// TIA Portal project "Aski-Otomasyonv2.2" (V16)

(* hardware
DEVICE "S71500/ET200MP station_1"  S7-1500 station
   slot 0: "Rail_0"  Rack  6ES7 590-1***0-0AA0
   slot 1: "PLC_8"  CPU 1511-1 PN  6ES7 511-1AK02-0AB0  V2.8
      slot 3: "CPU display_1"  6ES7591-1AA00-0AA0
      slot 32768: "PROFINET interface_1"  X1
         slot 32769: "Port_1"  X1 P1
         slot 32770: "Port_2"  X1 P2
      slot 34817: "Virtual CP interface port_1"  Virtual CP interface port  Virtual CP interface port
DEVICE "HMI_3"  KTP900 Basic PN
   slot 0: "HMI_3"  KTP900 Basic PN  6AV2 123-2JB03-0AX0  16.0.0.0
   slot 1: "HMI_RT_1"  KTP900 Basic PN  6AV2 123-2JB03-0AX0  16.0.0.0
   slot 5: "HMI_3.IE_CP_1"  PROFINET Interface  16.0.0.0
      slot 1: "PROFINET Interface_1"  PROFINET Interface
         slot 1: "Port_1"  Port
*)

// ===== PLC "PLC_8"  CPU 1511-1 PN =====

VAR_GLOBAL   // PLC tag table "Default tag table"
   "Start" AT %I0.0 : Bool;
   "Stop" AT %I0.1 : Bool;
   "sensor-HamSuKazan-alt" AT %I0.2 : Bool;
   "sensor-HamSuKazan-ust" AT %I0.3 : Bool;
   "sensor-TemizSuKazan-alt" AT %I0.4 : Bool;
   "sensor-TemizSuKazan-ust" AT %I0.5 : Bool;
   "aritmaMotor0" AT %Q0.0 : Bool;
   "aritmaMotor1" AT %Q0.1 : Bool;
   "aritmaMotor2" AT %Q0.2 : Bool;
   "motor-hamsu" AT %Q0.3 : Bool;
   "vana1-aritma0" AT %Q0.4 : Bool;
   "vana2-aritma0" AT %Q0.5 : Bool;
   "vana3-aritma0" AT %Q0.6 : Bool;
   "vana4-aritma0" AT %Q0.7 : Bool;
   "vana5-aritma0" AT %Q1.0 : Bool;
   "vana1-aritma1" AT %Q1.1 : Bool;
   "vana2-aritma1" AT %Q1.2 : Bool;
   "vana3-aritma1" AT %Q1.3 : Bool;
   "vana4-aritma1" AT %Q1.4 : Bool;
   "vana5-aritma1" AT %Q1.5 : Bool;
   "TimerTersYikama-aritma0" AT %T10 : Timer;
   "TimerDurulama-aritma0" AT %T11 : Timer;
   "Sistem" AT %Q1.6 : Bool;
   "TimerAritmaVana-aritma0" AT %T14 : Timer;
   "TimerTersYikamaVana-aritma0" AT %T15 : Timer;
   "TimerDurulamaVana-aritma0" AT %T16 : Timer;
   "TimerBypassVana-aritma0" AT %T17 : Timer;
   "TimerAritma-aritma0" AT %T18 : Timer;
   "sensor-SuCikisiVar" AT %I0.6 : Bool;
   "TimerMotor0Ariza" AT %T19 : Timer;
   "TimerMotor1Ariza" AT %T20 : Timer;
   "TimerMotor2Ariza" AT %T21 : Timer;
   "TimerAritmaVana-aritma1" AT %T22 : Timer;
   "TimerTersYikamaVana-aritma1" AT %T23 : Timer;
   "TimerDurulamaVana-aritma1" AT %T24 : Timer;
   "TimerBypassVana-aritma1" AT %T25 : Timer;
   "kuyuMotor" AT %I0.7 : Bool;
END_VAR

DATA_BLOCK "DBARITMA"   // DB1
{ S7_Optimized_Access := 'FALSE' }
VERSION : 0.1
   VAR
      "sure-Aritma" : S5Time := S5T#60s;
      "sure-TersYikama" : S5Time := S5T#20s;
      "sure-Durulama" : S5Time := S5T#10s;
      "sure-VanaDurumDegistirme" : S5Time := S5T#5s;
      "sure-MotorDegis" : Time := T#80s;
      "sure-MotorArizayaGec" : S5Time := S5T#5s;
      tesisDurumu : Byte := 0;
      toplamAritmaSayisi : Byte := 2;
      aritma0VanaKontrolDurum : Byte;
      aritma1VanaKontrolDurum : Byte;
      aritma0MotorCalisiyor : Bool;
      aritma1MotorCalisiyor : Bool;
      aritmaMotorCalisiyor : Bool;
      kalanZamanAritma : S5Time;
      kalanZamanTersYikama : S5Time;
      kalanZamanDurulama : S5Time;
      aritmaYapiliyor : Bool;
      tersYikamaYapiliyor : Bool;
      durulamaYapiliyor : Bool;
      aritmaMotor0Durum : Byte;
      aritmaMotor1Durum : Byte;
      aritmaMotor2Durum : Byte;
      kuyuMotorDurum : Byte := 0;
      durumKalanSure : Word := 1;
      temizsuSeviye : Byte := 45;
      hamsuSeviye : Byte := 92;
      arizaDurumu : Byte := 0;
      Adi : String := 'Deneme Tesis';
      temizsuDepoDoldur : Bool;
      "hmi-start" : Bool;
      "hmi-stop" : Bool;
      "hmi-aritmaSure" : Byte;
      "hmi-TersYikamaSure" : Byte;
      "hmi-DurulamaSure" : Byte;
      "hmi-VanaBeklemeSure" : Byte;
      "hmi-YaslandirmaSure" : Byte := 20;
      "hmi-TersYikamaYap" : Bool;
   END_VAR
BEGIN
END_DATA_BLOCK

DATA_BLOCK "FB-aritma0VanaKontrol_DB"   // DB2
{ S7_Optimized_Access := 'TRUE' }
VERSION : 0.1
// stored: InstanceOfName FB-aritmaVanaKontrol
"FB-aritmaVanaKontrol"
BEGIN
END_DATA_BLOCK

DATA_BLOCK "sistemDurum-Zamanlayici_DB"   // DB3
{ S7_Optimized_Access := 'TRUE' }
VERSION : 0.1
// stored: InstanceOfName aritmaDurum-Zamanlayici
"aritmaDurum-Zamanlayici"
BEGIN
END_DATA_BLOCK

DATA_BLOCK "aritmaMotorKontrol-Yaslandirma-Ariza_DB"   // DB4
{ S7_Optimized_Access := 'TRUE' }
VERSION : 0.1
// stored: InstanceOfName aritmaMotorKontrol-Yaslandirma-Ariza
"aritmaMotorKontrol-Yaslandirma-Ariza"
BEGIN
END_DATA_BLOCK

DATA_BLOCK "FB-aritma1VanaKontrol_DB"   // DB6
{ S7_Optimized_Access := 'TRUE' }
VERSION : 0.1
// stored: InstanceOfName FB-aritmaVanaKontrol
"FB-aritmaVanaKontrol"
BEGIN
END_DATA_BLOCK

DATA_BLOCK "TemizSuDepoSeviyeKonrolcusu"   // DB7
{ S7_Optimized_Access := 'TRUE' }
VERSION : 0.1
// stored: InstanceOfName depoSeviyeKonrolcusu
"depoSeviyeKonrolcusu"
BEGIN
END_DATA_BLOCK

DATA_BLOCK "HamSuDepoSeviyeKonrolcusu"   // DB8
{ S7_Optimized_Access := 'TRUE' }
VERSION : 0.1
// stored: InstanceOfName depoSeviyeKonrolcusu
"depoSeviyeKonrolcusu"
BEGIN
END_DATA_BLOCK

// folder: System blocks/Program resources

DATA_BLOCK "timerMotorDegistirme"   // DB5
{ S7_Optimized_Access := 'TRUE' }
AUTHOR : Simatic
FAMILY : IEC
NAME : IEC_TMR
VERSION : 1.0
// stored: InstanceOfName IEC_TIMER
"IEC_TIMER"
BEGIN
END_DATA_BLOCK

// folder: (top level)

FUNCTION_BLOCK "FB-aritmaVanaKontrol"   // FB1, LAD
{ S7_Optimized_Access := 'TRUE' }
VERSION : 0.1
   VAR_INPUT
      Sistem : Bool;
      timerAritmaVana : Timer;
      timerTersYikamaVana : Timer;
      timerDurulamaVana : Timer;
      timerBypassVana : Timer;
      "sure-VanaDurumDegisim" : S5Time;
      aritmaDurumu : Byte;
   END_VAR
   VAR_OUTPUT
      V1 : Bool;
      V2 : Bool;
      V3 : Bool;
      V4 : Bool;
      V5 : Bool;
      "aritma-motoru-Calistir" : Bool;
   END_VAR
   VAR
      aritmaDurumunaGec : Bool;
      tersYikamaDurumunaGec : Bool;
      durulamaDurumunaGec : Bool;
      bypassDurumunaGec : Bool;
      "motoruAktifEt-Aritma" : Bool;
      "motoruAktifEt-TersYikama" : Bool;
      "motoruAktifEt-Durulama" : Bool;
      "motoruAktifEt-Bypass" : Bool;
   END_VAR
   VAR_TEMP   // added for the SCL form of the ladder/FBD networks
      _w1 : Bool;
      _w2 : Bool;
      _w3 : Bool;
      _w4 : Bool;
      _s5time1 : S5Time;
   END_VAR
BEGIN

REGION Network 1: Vana Durum ayarlamaları
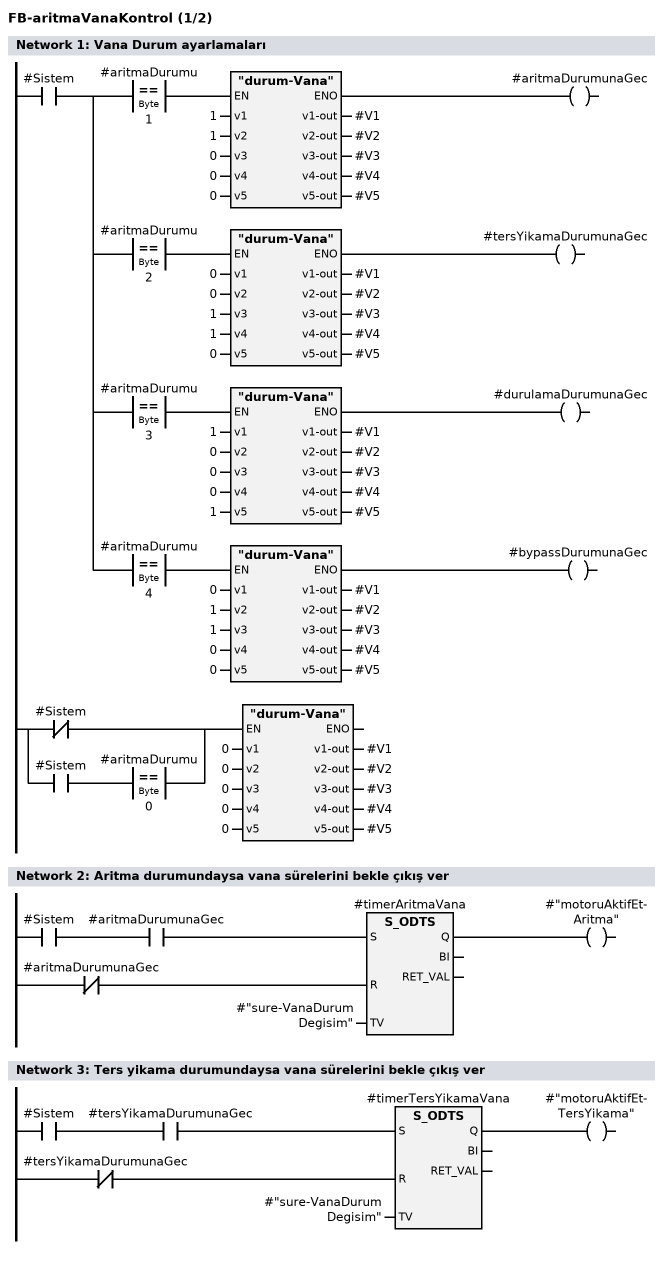
   RUNG wire#powerrail
      Contact( #Sistem )
      wire#w1
      { S7_Templates := "SrcType := Byte" } EQ_Contact(in1 := #aritmaDurumu, in2 := 1)
      "durum-Vana"(v1 := 1, v2 := 1, v3 := 0, v4 := 0, v5 := 0, "v1-out" => #V1, "v2-out" => #V2, "v3-out" => #V3, "v4-out" => #V4, "v5-out" => #V5)
      Coil( #aritmaDurumunaGec )
   END_RUNG
   RUNG wire#w1
      { S7_Templates := "SrcType := Byte" } EQ_Contact(in1 := #aritmaDurumu, in2 := 2)
      "durum-Vana"(v1 := 0, v2 := 0, v3 := 1, v4 := 1, v5 := 0, "v1-out" => #V1, "v2-out" => #V2, "v3-out" => #V3, "v4-out" => #V4, "v5-out" => #V5)
      Coil( #tersYikamaDurumunaGec )
   END_RUNG
   RUNG wire#w1
      { S7_Templates := "SrcType := Byte" } EQ_Contact(in1 := #aritmaDurumu, in2 := 3)
      "durum-Vana"(v1 := 1, v2 := 0, v3 := 0, v4 := 0, v5 := 1, "v1-out" => #V1, "v2-out" => #V2, "v3-out" => #V3, "v4-out" => #V4, "v5-out" => #V5)
      Coil( #durulamaDurumunaGec )
   END_RUNG
   RUNG wire#w1
      { S7_Templates := "SrcType := Byte" } EQ_Contact(in1 := #aritmaDurumu, in2 := 4)
      "durum-Vana"(v1 := 0, v2 := 1, v3 := 1, v4 := 0, v5 := 0, "v1-out" => #V1, "v2-out" => #V2, "v3-out" => #V3, "v4-out" => #V4, "v5-out" => #V5)
      Coil( #bypassDurumunaGec )
   END_RUNG
   RUNG wire#powerrail
      I_Contact( #Sistem )
      wire#w2
      "durum-Vana"(v1 := 0, v2 := 0, v3 := 0, v4 := 0, v5 := 0, "v1-out" => #V1, "v2-out" => #V2, "v3-out" => #V3, "v4-out" => #V4, "v5-out" => #V5)
   END_RUNG
   RUNG wire#powerrail
      Contact( #Sistem )
      { S7_Templates := "SrcType := Byte" } EQ_Contact(in1 := #aritmaDurumu, in2 := 0)
   END_RUNG wire#w2
   // the same network as SCL:
   "durum-Vana"(EN := #Sistem AND (#aritmaDurumu = 1),
                v1 := 1,
                v2 := 1,
                v3 := 0,
                v4 := 0,
                v5 := 0,
                "v1-out" => #V1,
                "v2-out" => #V2,
                "v3-out" => #V3,
                "v4-out" => #V4,
                "v5-out" => #V5,
                ENO => #_w1);
   #aritmaDurumunaGec := #_w1;
   "durum-Vana"(EN := #Sistem AND (#aritmaDurumu = 2),
                v1 := 0,
                v2 := 0,
                v3 := 1,
                v4 := 1,
                v5 := 0,
                "v1-out" => #V1,
                "v2-out" => #V2,
                "v3-out" => #V3,
                "v4-out" => #V4,
                "v5-out" => #V5,
                ENO => #_w2);
   #tersYikamaDurumunaGec := #_w2;
   "durum-Vana"(EN := #Sistem AND (#aritmaDurumu = 3),
                v1 := 1,
                v2 := 0,
                v3 := 0,
                v4 := 0,
                v5 := 1,
                "v1-out" => #V1,
                "v2-out" => #V2,
                "v3-out" => #V3,
                "v4-out" => #V4,
                "v5-out" => #V5,
                ENO => #_w3);
   #durulamaDurumunaGec := #_w3;
   "durum-Vana"(EN := #Sistem AND (#aritmaDurumu = 4),
                v1 := 0,
                v2 := 1,
                v3 := 1,
                v4 := 0,
                v5 := 0,
                "v1-out" => #V1,
                "v2-out" => #V2,
                "v3-out" => #V3,
                "v4-out" => #V4,
                "v5-out" => #V5,
                ENO => #_w4);
   #bypassDurumunaGec := #_w4;
   IF NOT #Sistem OR (#Sistem AND (#aritmaDurumu = 0)) THEN
       "durum-Vana"(v1 := 0,
                    v2 := 0,
                    v3 := 0,
                    v4 := 0,
                    v5 := 0,
                    "v1-out" => #V1,
                    "v2-out" => #V2,
                    "v3-out" => #V3,
                    "v4-out" => #V4,
                    "v5-out" => #V5);
   END_IF;
END_REGION

REGION Network 2: Aritma durumundaysa vana sürelerini bekle çıkış ver
   RUNG wire#powerrail
      Contact( #Sistem )
      Contact( #aritmaDurumunaGec )
      S_ODTS(T_NO := #timerAritmaVana, R := wire#w1, TV := #"sure-VanaDurumDegisim", BI =>, RET_VAL =>)
      Coil( #"motoruAktifEt-Aritma" )
   END_RUNG
   RUNG wire#powerrail
      I_Contact( #aritmaDurumunaGec )
   END_RUNG wire#w1
   // the same network as SCL:
   #_s5time1 := S_ODTS(T_NO := #timerAritmaVana,
                       S := #Sistem AND #aritmaDurumunaGec,
                       R := NOT #aritmaDurumunaGec,
                       TV := #"sure-VanaDurumDegisim",
                       Q => #_w1);
   #"motoruAktifEt-Aritma" := #_w1;
END_REGION

REGION Network 3: Ters yikama durumundaysa vana sürelerini bekle çıkış ver
   RUNG wire#powerrail
      Contact( #Sistem )
      Contact( #tersYikamaDurumunaGec )
      S_ODTS(T_NO := #timerTersYikamaVana, R := wire#w1, TV := #"sure-VanaDurumDegisim", BI =>, RET_VAL =>)
      Coil( #"motoruAktifEt-TersYikama" )
   END_RUNG
   RUNG wire#powerrail
      I_Contact( #tersYikamaDurumunaGec )
   END_RUNG wire#w1
   // the same network as SCL:
   #_s5time1 := S_ODTS(T_NO := #timerTersYikamaVana,
                       S := #Sistem AND #tersYikamaDurumunaGec,
                       R := NOT #tersYikamaDurumunaGec,
                       TV := #"sure-VanaDurumDegisim",
                       Q => #_w1);
   #"motoruAktifEt-TersYikama" := #_w1;
END_REGION

REGION Network 4: Durulama durumundaysa vana sürelerini bekle çıkış ver
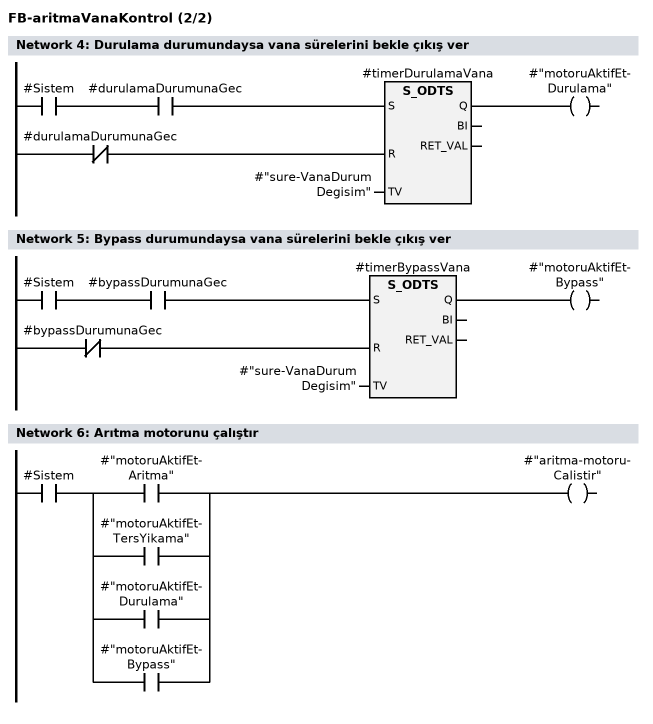
   RUNG wire#powerrail
      Contact( #Sistem )
      Contact( #durulamaDurumunaGec )
      S_ODTS(T_NO := #timerDurulamaVana, R := wire#w1, TV := #"sure-VanaDurumDegisim", BI =>, RET_VAL =>)
      Coil( #"motoruAktifEt-Durulama" )
   END_RUNG
   RUNG wire#powerrail
      I_Contact( #durulamaDurumunaGec )
   END_RUNG wire#w1
   // the same network as SCL:
   #_s5time1 := S_ODTS(T_NO := #timerDurulamaVana,
                       S := #Sistem AND #durulamaDurumunaGec,
                       R := NOT #durulamaDurumunaGec,
                       TV := #"sure-VanaDurumDegisim",
                       Q => #_w1);
   #"motoruAktifEt-Durulama" := #_w1;
END_REGION

REGION Network 5: Bypass durumundaysa vana sürelerini bekle çıkış ver
   RUNG wire#powerrail
      Contact( #Sistem )
      Contact( #bypassDurumunaGec )
      S_ODTS(T_NO := #timerBypassVana, R := wire#w1, TV := #"sure-VanaDurumDegisim", BI =>, RET_VAL =>)
      Coil( #"motoruAktifEt-Bypass" )
   END_RUNG
   RUNG wire#powerrail
      I_Contact( #bypassDurumunaGec )
   END_RUNG wire#w1
   // the same network as SCL:
   #_s5time1 := S_ODTS(T_NO := #timerBypassVana,
                       S := #Sistem AND #bypassDurumunaGec,
                       R := NOT #bypassDurumunaGec,
                       TV := #"sure-VanaDurumDegisim",
                       Q => #_w1);
   #"motoruAktifEt-Bypass" := #_w1;
END_REGION

REGION Network 6: Arıtma motorunu çalıştır
   RUNG wire#powerrail
      Contact( #Sistem )
      wire#w1
      Contact( #"motoruAktifEt-Aritma" )
      wire#w2
      Coil( #"aritma-motoru-Calistir" )
   END_RUNG
   RUNG wire#w1
      Contact( #"motoruAktifEt-TersYikama" )
   END_RUNG wire#w2
   RUNG wire#w1
      Contact( #"motoruAktifEt-Durulama" )
   END_RUNG wire#w2
   RUNG wire#w1
      Contact( #"motoruAktifEt-Bypass" )
   END_RUNG wire#w2
   // the same network as SCL:
   #"aritma-motoru-Calistir" := #Sistem AND (#"motoruAktifEt-Aritma" OR #"motoruAktifEt-TersYikama" OR #"motoruAktifEt-Durulama" OR #"motoruAktifEt-Bypass");
END_REGION
END_FUNCTION_BLOCK

FUNCTION_BLOCK "aritmaDurum-Zamanlayici"   // FB2, LAD
{ S7_Optimized_Access := 'TRUE' }
VERSION : 0.1
   VAR_INPUT
      sistem : Bool;
      "motor-aritma-calisiyor" : Bool;
      sureAritma : S5Time;
      sureTersYikama : S5Time;
      sureDurulama : S5Time;
      timerAritma : Timer;
      timerTersYikama : Timer;
      timerDurulama : Timer;
      maxDurumSayisi : Byte;
   END_VAR
   VAR_OUTPUT
      kalanZamanAritma : S5Time;
      kalanZamanTersYikama : S5Time;
      kalanZamanDurulama : S5Time;
      durulamaYapiliyorBilgisi : Bool;
      tersYikamaYapiliyorBilgisi : Bool;
      aritmaYapiliyorBilgisi : Bool;
   END_VAR
   VAR_IN_OUT
      tesisDurumu : Byte;
   END_VAR
   VAR_TEMP
      aritmaYapiliyor : Bool;
      tersYikamaYapiliyor : Bool;
      durulamaYapiliyor : Bool;
   END_VAR
   VAR CONSTANT
      durumBuffer : Byte;
   END_VAR
   VAR_TEMP   // added for the SCL form of the ladder/FBD networks
      _w1 : Bool;
      _s5time1 : S5Time;
   END_VAR
BEGIN

REGION Network 1: Durum ayarlamaları 2 arıtmalı için*
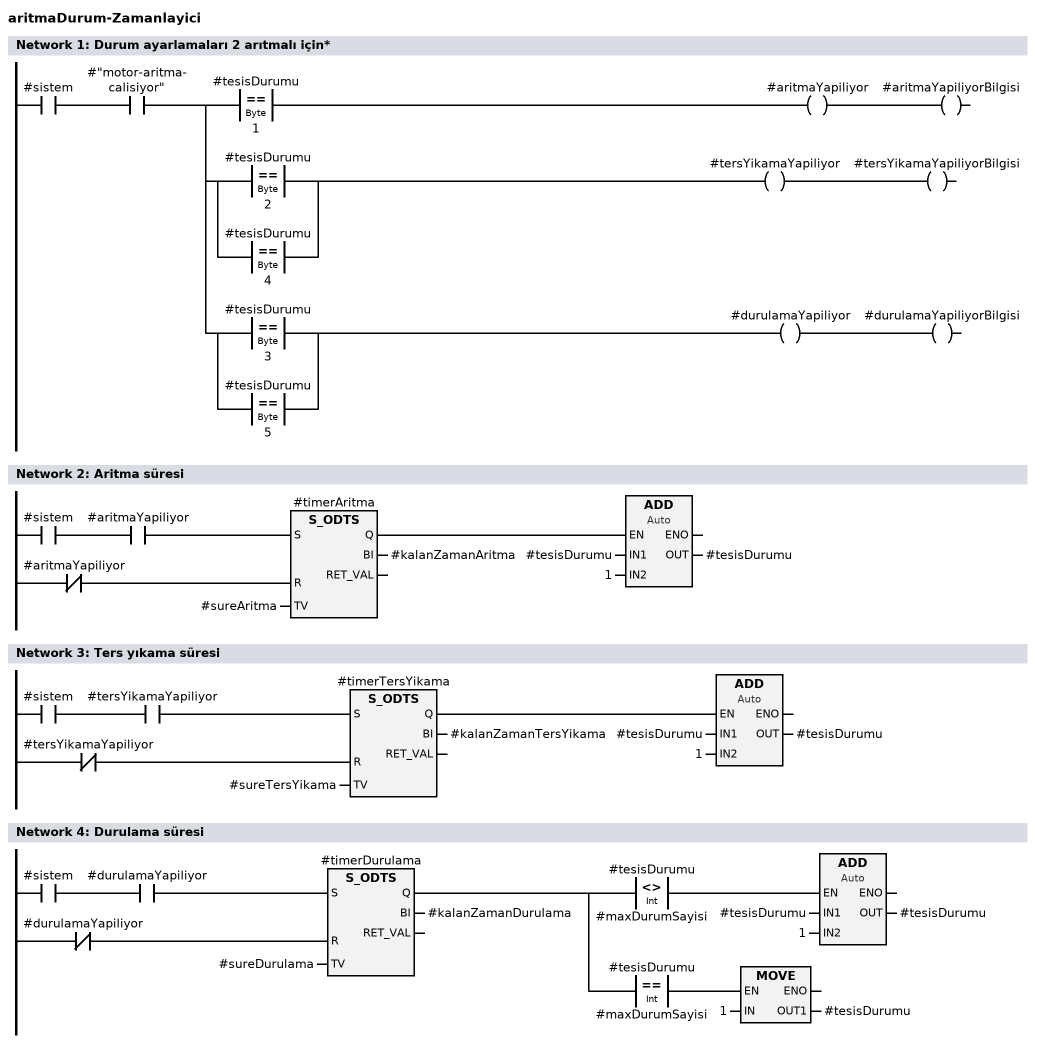
   RUNG wire#powerrail
      Contact( #sistem )
      Contact( #"motor-aritma-calisiyor" )
      wire#w1
      { S7_Templates := "SrcType := Byte" } EQ_Contact(in1 := #tesisDurumu, in2 := 1)
      Coil( #aritmaYapiliyor )
      Coil( #aritmaYapiliyorBilgisi )
   END_RUNG
   RUNG wire#w1
      { S7_Templates := "SrcType := Byte" } EQ_Contact(in1 := #tesisDurumu, in2 := 2)
      wire#w2
      Coil( #tersYikamaYapiliyor )
      Coil( #tersYikamaYapiliyorBilgisi )
   END_RUNG
   RUNG wire#w1
      { S7_Templates := "SrcType := Byte" } EQ_Contact(in1 := #tesisDurumu, in2 := 4)
   END_RUNG wire#w2
   RUNG wire#w1
      { S7_Templates := "SrcType := Byte" } EQ_Contact(in1 := #tesisDurumu, in2 := 3)
      wire#w3
      Coil( #durulamaYapiliyor )
      Coil( #durulamaYapiliyorBilgisi )
   END_RUNG
   RUNG wire#w1
      { S7_Templates := "SrcType := Byte" } EQ_Contact(in1 := #tesisDurumu, in2 := 5)
   END_RUNG wire#w3
   // the same network as SCL:
   #_w1 := #sistem AND #"motor-aritma-calisiyor";
   #aritmaYapiliyor := #_w1 AND (#tesisDurumu = 1);
   #aritmaYapiliyorBilgisi := #aritmaYapiliyor;
   #tersYikamaYapiliyor := #_w1 AND ((#tesisDurumu = 2) OR (#tesisDurumu = 4));
   #tersYikamaYapiliyorBilgisi := #tersYikamaYapiliyor;
   #durulamaYapiliyor := #_w1 AND ((#tesisDurumu = 3) OR (#tesisDurumu = 5));
   #durulamaYapiliyorBilgisi := #durulamaYapiliyor;
END_REGION

REGION Network 2: Aritma süresi
   RUNG wire#powerrail
      Contact( #sistem )
      Contact( #aritmaYapiliyor )
      S_ODTS(T_NO := #timerAritma, R := wire#w1, TV := #sureAritma, BI => #kalanZamanAritma, RET_VAL =>)
      Add(in1 := #tesisDurumu, in2 := 1, out => #tesisDurumu)
   END_RUNG
   RUNG wire#powerrail
      I_Contact( #aritmaYapiliyor )
   END_RUNG wire#w1
   // the same network as SCL:
   #_s5time1 := S_ODTS(T_NO := #timerAritma,
                       S := #sistem AND #aritmaYapiliyor,
                       R := NOT #aritmaYapiliyor,
                       TV := #sureAritma,
                       Q => #_w1,
                       BI => #kalanZamanAritma);
   IF #_w1 THEN #tesisDurumu := #tesisDurumu + 1; END_IF;
END_REGION

REGION Network 3: Ters yıkama süresi
   RUNG wire#powerrail
      Contact( #sistem )
      Contact( #tersYikamaYapiliyor )
      S_ODTS(T_NO := #timerTersYikama, R := wire#w1, TV := #sureTersYikama, BI => #kalanZamanTersYikama, RET_VAL =>)
      Add(in1 := #tesisDurumu, in2 := 1, out => #tesisDurumu)
   END_RUNG
   RUNG wire#powerrail
      I_Contact( #tersYikamaYapiliyor )
   END_RUNG wire#w1
   // the same network as SCL:
   #_s5time1 := S_ODTS(T_NO := #timerTersYikama,
                       S := #sistem AND #tersYikamaYapiliyor,
                       R := NOT #tersYikamaYapiliyor,
                       TV := #sureTersYikama,
                       Q => #_w1,
                       BI => #kalanZamanTersYikama);
   IF #_w1 THEN #tesisDurumu := #tesisDurumu + 1; END_IF;
END_REGION

REGION Network 4: Durulama süresi
   RUNG wire#powerrail
      Contact( #sistem )
      Contact( #durulamaYapiliyor )
      S_ODTS(T_NO := #timerDurulama, R := wire#w1, TV := #sureDurulama, BI => #kalanZamanDurulama, RET_VAL =>)
      wire#w2
      { S7_Templates := "SrcType := Int" } NE_Contact(in1 := #tesisDurumu, in2 := #maxDurumSayisi)
      Add(in1 := #tesisDurumu, in2 := 1, out => #tesisDurumu)
   END_RUNG
   RUNG wire#powerrail
      I_Contact( #durulamaYapiliyor )
   END_RUNG wire#w1
   RUNG wire#w2
      { S7_Templates := "SrcType := Int" } EQ_Contact(in1 := #tesisDurumu, in2 := #maxDurumSayisi)
      Move(in := 1, out1 => #tesisDurumu)
   END_RUNG
   // the same network as SCL:
   #_s5time1 := S_ODTS(T_NO := #timerDurulama,
                       S := #sistem AND #durulamaYapiliyor,
                       R := NOT #durulamaYapiliyor,
                       TV := #sureDurulama,
                       Q => #_w1,
                       BI => #kalanZamanDurulama);
   IF #_w1 AND (#tesisDurumu <> #maxDurumSayisi) THEN #tesisDurumu := #tesisDurumu + 1; END_IF;
   IF #_w1 AND (#tesisDurumu = #maxDurumSayisi) THEN #tesisDurumu := 1; END_IF;
END_REGION
END_FUNCTION_BLOCK

FUNCTION_BLOCK "aritmaMotorKontrol-Yaslandirma-Ariza"   // FB3, LAD
{ S7_Optimized_Access := 'TRUE' }
VERSION : 0.1
   VAR_INPUT
      sistem : Bool;
      "motor-calistir" : Bool;
      "sensor-su-cikisi-var" : Bool;
      timerMotor0Ariza : Timer;
      timerMotor1Ariza : Timer;
      timerMotor2Ariza : Timer;
      sureMotorDegis : Time;
      sureArizayaGec : S5Time;
   END_VAR
   VAR_OUTPUT
      aritmaMotor0 : Bool;
      aritmaMotor1 : Bool;
      aritmaMotor2 : Bool;
      motor0Durum : Byte;
      motor1Durum : Byte;
      motor2Durum : Byte;
      sistemStop : Bool;
   END_VAR
   VAR
      motorSirasi : Int;
      yk0 : Bool;
      yk1 : Bool;
      yk2 : Bool;
   END_VAR
   VAR_TEMP   // added for the SCL form of the ladder/FBD networks
      _w1 : Bool;
      _w2 : Bool;
      _s5time1 : S5Time;
      _w3 : Bool;
      _s5time2 : S5Time;
      _w4 : Bool;
      _s5time3 : S5Time;
   END_VAR
BEGIN

REGION Network 1: Motor Sırasını kontrol et ve Sıradaki motoru aktif et
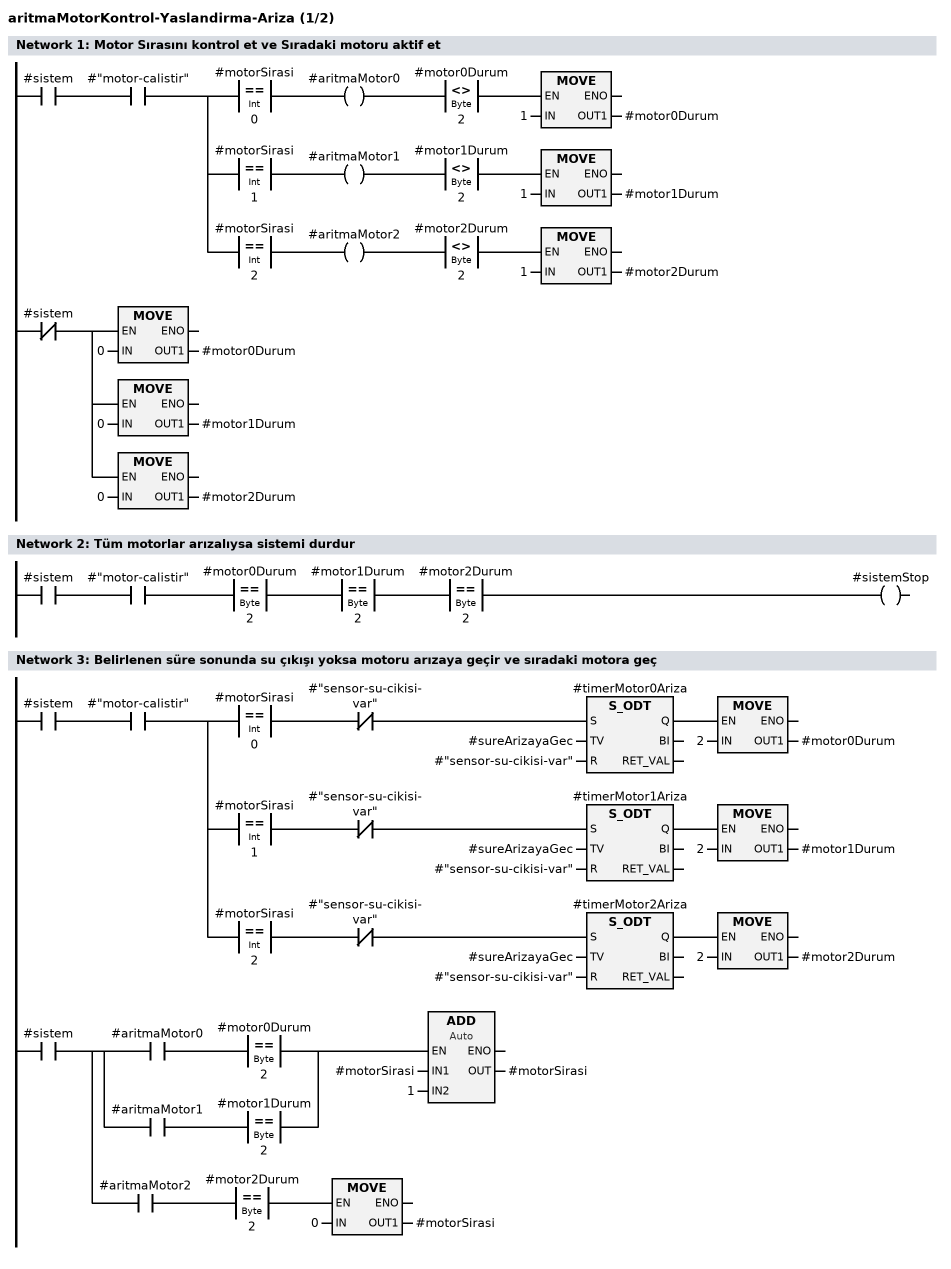
   RUNG wire#powerrail
      Contact( #sistem )
      Contact( #"motor-calistir" )
      wire#w1
      { S7_Templates := "SrcType := Int" } EQ_Contact(in1 := #motorSirasi, in2 := 0)
      Coil( #aritmaMotor0 )
      { S7_Templates := "SrcType := Byte" } NE_Contact(in1 := #motor0Durum, in2 := 2)
      Move(in := 1, out1 => #motor0Durum)
   END_RUNG
   RUNG wire#w1
      { S7_Templates := "SrcType := Int" } EQ_Contact(in1 := #motorSirasi, in2 := 1)
      Coil( #aritmaMotor1 )
      { S7_Templates := "SrcType := Byte" } NE_Contact(in1 := #motor1Durum, in2 := 2)
      Move(in := 1, out1 => #motor1Durum)
   END_RUNG
   RUNG wire#w1
      { S7_Templates := "SrcType := Int" } EQ_Contact(in1 := #motorSirasi, in2 := 2)
      Coil( #aritmaMotor2 )
      { S7_Templates := "SrcType := Byte" } NE_Contact(in1 := #motor2Durum, in2 := 2)
      Move(in := 1, out1 => #motor2Durum)
   END_RUNG
   RUNG wire#powerrail
      I_Contact( #sistem )
      wire#w2
      Move(in := 0, out1 => #motor0Durum)
   END_RUNG
   RUNG wire#w2
      Move(in := 0, out1 => #motor1Durum)
   END_RUNG
   RUNG wire#w2
      Move(in := 0, out1 => #motor2Durum)
   END_RUNG
   // the same network as SCL:
   #_w1 := #sistem AND #"motor-calistir";
   #aritmaMotor0 := #_w1 AND (#motorSirasi = 0);
   IF #aritmaMotor0 AND (#motor0Durum <> 2) THEN #motor0Durum := 1; END_IF;
   #aritmaMotor1 := #_w1 AND (#motorSirasi = 1);
   IF #aritmaMotor1 AND (#motor1Durum <> 2) THEN #motor1Durum := 1; END_IF;
   #aritmaMotor2 := #_w1 AND (#motorSirasi = 2);
   IF #aritmaMotor2 AND (#motor2Durum <> 2) THEN #motor2Durum := 1; END_IF;
   IF NOT #sistem THEN
       #motor0Durum := 0;
       #motor1Durum := 0;
       #motor2Durum := 0;
   END_IF;
END_REGION

REGION Network 2: Tüm motorlar arızalıysa sistemi durdur
   RUNG wire#powerrail
      Contact( #sistem )
      Contact( #"motor-calistir" )
      { S7_Templates := "SrcType := Byte" } EQ_Contact(in1 := #motor0Durum, in2 := 2)
      { S7_Templates := "SrcType := Byte" } EQ_Contact(in1 := #motor1Durum, in2 := 2)
      { S7_Templates := "SrcType := Byte" } EQ_Contact(in1 := #motor2Durum, in2 := 2)
      Coil( #sistemStop )
   END_RUNG
   // the same network as SCL:
   #sistemStop := #sistem AND #"motor-calistir" AND (#motor0Durum = 2) AND (#motor1Durum = 2) AND (#motor2Durum = 2);
END_REGION

REGION Network 3: Belirlenen süre sonunda su çıkışı yoksa motoru arızaya geçir ve sıradaki motora geç
   RUNG wire#powerrail
      Contact( #sistem )
      Contact( #"motor-calistir" )
      wire#w1
      { S7_Templates := "SrcType := Int" } EQ_Contact(in1 := #motorSirasi, in2 := 0)
      I_Contact( #"sensor-su-cikisi-var" )
      S_ODT(T_NO := #timerMotor0Ariza, TV := #sureArizayaGec, R := #"sensor-su-cikisi-var", BI =>, RET_VAL =>)
      Move(in := 2, out1 => #motor0Durum)
   END_RUNG
   RUNG wire#w1
      { S7_Templates := "SrcType := Int" } EQ_Contact(in1 := #motorSirasi, in2 := 1)
      I_Contact( #"sensor-su-cikisi-var" )
      S_ODT(T_NO := #timerMotor1Ariza, TV := #sureArizayaGec, R := #"sensor-su-cikisi-var", BI =>, RET_VAL =>)
      Move(in := 2, out1 => #motor1Durum)
   END_RUNG
   RUNG wire#w1
      { S7_Templates := "SrcType := Int" } EQ_Contact(in1 := #motorSirasi, in2 := 2)
      I_Contact( #"sensor-su-cikisi-var" )
      S_ODT(T_NO := #timerMotor2Ariza, TV := #sureArizayaGec, R := #"sensor-su-cikisi-var", BI =>, RET_VAL =>)
      Move(in := 2, out1 => #motor2Durum)
   END_RUNG
   RUNG wire#powerrail
      Contact( #sistem )
      wire#w2
      Contact( #aritmaMotor0 )
      { S7_Templates := "SrcType := Byte" } EQ_Contact(in1 := #motor0Durum, in2 := 2)
      wire#w3
      Add(in1 := #motorSirasi, in2 := 1, out => #motorSirasi)
   END_RUNG
   RUNG wire#w2
      Contact( #aritmaMotor1 )
      { S7_Templates := "SrcType := Byte" } EQ_Contact(in1 := #motor1Durum, in2 := 2)
   END_RUNG wire#w3
   RUNG wire#w2
      Contact( #aritmaMotor2 )
      { S7_Templates := "SrcType := Byte" } EQ_Contact(in1 := #motor2Durum, in2 := 2)
      Move(in := 0, out1 => #motorSirasi)
   END_RUNG
   // the same network as SCL:
   #_w1 := #sistem AND #"motor-calistir";
   #_s5time1 := S_ODT(T_NO := #timerMotor0Ariza,
                      S := #_w1 AND (#motorSirasi = 0) AND NOT #"sensor-su-cikisi-var",
                      TV := #sureArizayaGec,
                      R := #"sensor-su-cikisi-var",
                      Q => #_w2);
   IF #_w2 THEN #motor0Durum := 2; END_IF;
   #_s5time2 := S_ODT(T_NO := #timerMotor1Ariza,
                      S := #_w1 AND (#motorSirasi = 1) AND NOT #"sensor-su-cikisi-var",
                      TV := #sureArizayaGec,
                      R := #"sensor-su-cikisi-var",
                      Q => #_w3);
   IF #_w3 THEN #motor1Durum := 2; END_IF;
   #_s5time3 := S_ODT(T_NO := #timerMotor2Ariza,
                      S := #_w1 AND (#motorSirasi = 2) AND NOT #"sensor-su-cikisi-var",
                      TV := #sureArizayaGec,
                      R := #"sensor-su-cikisi-var",
                      Q => #_w4);
   IF #_w4 THEN #motor2Durum := 2; END_IF;
   IF #sistem AND ((#aritmaMotor0 AND (#motor0Durum = 2)) OR (#aritmaMotor1 AND (#motor1Durum = 2))) THEN
       #motorSirasi := #motorSirasi + 1;
   END_IF;
   IF #sistem AND #aritmaMotor2 AND (#motor2Durum = 2) THEN #motorSirasi := 0; END_IF;
END_REGION

REGION Network 4: Belirlenen süre sonunda Sıradaki motora geç
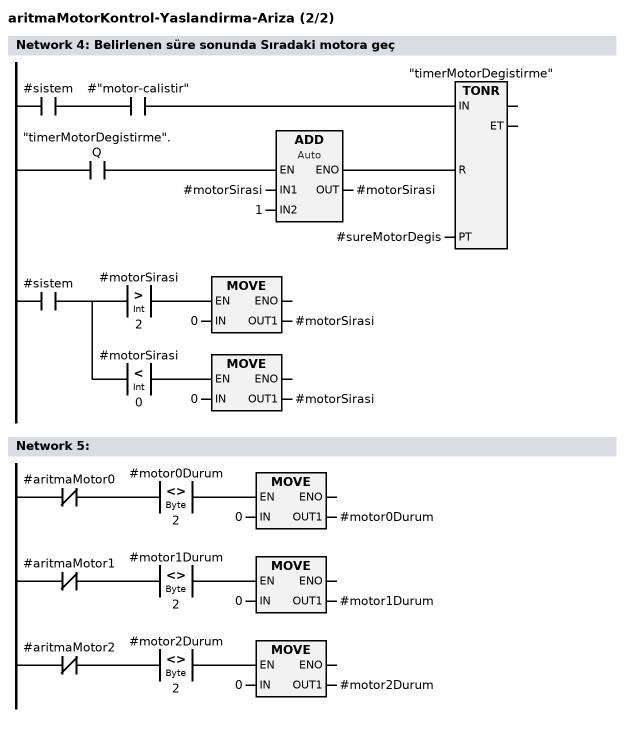
   IF "timerMotorDegistirme".Q THEN #motorSirasi := #motorSirasi + 1; END_IF;
   "timerMotorDegistirme".TONR(IN := #sistem AND #"motor-calistir",
                           R := "timerMotorDegistirme".Q,
                           PT := #sureMotorDegis);
   IF #sistem AND (#motorSirasi > 2) THEN #motorSirasi := 0; END_IF;
   IF #sistem AND (#motorSirasi < 0) THEN #motorSirasi := 0; END_IF;
END_REGION

REGION Network 5
   RUNG wire#powerrail
      I_Contact( #aritmaMotor0 )
      { S7_Templates := "SrcType := Byte" } NE_Contact(in1 := #motor0Durum, in2 := 2)
      Move(in := 0, out1 => #motor0Durum)
   END_RUNG
   RUNG wire#powerrail
      I_Contact( #aritmaMotor1 )
      { S7_Templates := "SrcType := Byte" } NE_Contact(in1 := #motor1Durum, in2 := 2)
      Move(in := 0, out1 => #motor1Durum)
   END_RUNG
   RUNG wire#powerrail
      I_Contact( #aritmaMotor2 )
      { S7_Templates := "SrcType := Byte" } NE_Contact(in1 := #motor2Durum, in2 := 2)
      Move(in := 0, out1 => #motor2Durum)
   END_RUNG
   // the same network as SCL:
   IF NOT #aritmaMotor0 AND (#motor0Durum <> 2) THEN #motor0Durum := 0; END_IF;
   IF NOT #aritmaMotor1 AND (#motor1Durum <> 2) THEN #motor1Durum := 0; END_IF;
   IF NOT #aritmaMotor2 AND (#motor2Durum <> 2) THEN #motor2Durum := 0; END_IF;
END_REGION
END_FUNCTION_BLOCK

FUNCTION_BLOCK "depoSeviyeKonrolcusu"   // FB4, LAD
{ S7_Optimized_Access := 'TRUE' }
VERSION : 0.1
   VAR_INPUT
      sistem : Bool;
      depoAltSeviyeSensor : Bool;
      depoUstSeviyeSensor : Bool;
      anlikSuGirisDebisi : Int;
      anlikSuCikisDebisi : Int;
      depoAltSensorKonumu : Int;
      depoUstSensorKonumu : Int;
   END_VAR
   VAR_OUTPUT
      depoyuDoldur : Bool;
      depoSeviyesi : Int;
   END_VAR
   VAR
      mdepoyuDoldur : Bool;
   END_VAR
BEGIN

REGION Network 1: Alt sensör su algılamadığında depoyu üst sensör görene kadar doldur.
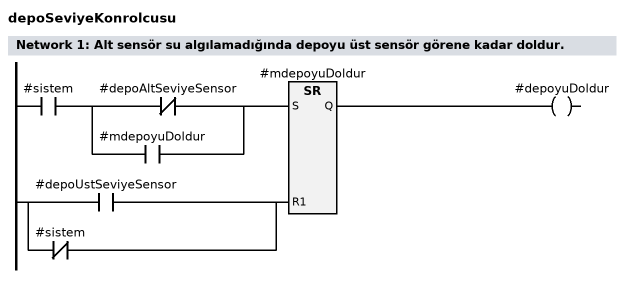
   RUNG wire#powerrail
      Contact( #sistem )
      wire#w1
      I_Contact( #depoAltSeviyeSensor )
      wire#w2
      S_SR(operand := #mdepoyuDoldur, r1 := wire#w3)
      Coil( #depoyuDoldur )
   END_RUNG
   RUNG wire#w1
      Contact( #mdepoyuDoldur )
   END_RUNG wire#w2
   RUNG wire#powerrail
      Contact( #depoUstSeviyeSensor )
   END_RUNG wire#w3
   RUNG wire#powerrail
      I_Contact( #sistem )
   END_RUNG wire#w3
   // the same network as SCL:
   IF #sistem AND (NOT #depoAltSeviyeSensor OR #mdepoyuDoldur) THEN
       #mdepoyuDoldur := TRUE;   // SR flip-flop
   END_IF;
   IF #depoUstSeviyeSensor OR NOT #sistem THEN #mdepoyuDoldur := FALSE; END_IF;
   #depoyuDoldur := #mdepoyuDoldur;
END_REGION

REGION Network 2: Depodaki su seviyesini yaklaşık olarak hesapla
END_REGION
END_FUNCTION_BLOCK

FUNCTION "durum-Vana" : Void   // FC1, LAD
{ S7_Optimized_Access := 'TRUE' }
VERSION : 0.1
   VAR_INPUT
      v1 : Bool;
      v2 : Bool;
      v3 : Bool;
      v4 : Bool;
      v5 : Bool;
   END_VAR
   VAR_OUTPUT
      "v1-out" : Bool;
      "v2-out" : Bool;
      "v3-out" : Bool;
      "v4-out" : Bool;
      "v5-out" : Bool;
   END_VAR
   VAR_TEMP
      "m_v1-out" : Bool;
      "m_v2-out" : Bool;
      "m_v3-out" : Bool;
      "m_v4-out" : Bool;
      "m_v5-out" : Bool;
   END_VAR
BEGIN

REGION Network 1: V1
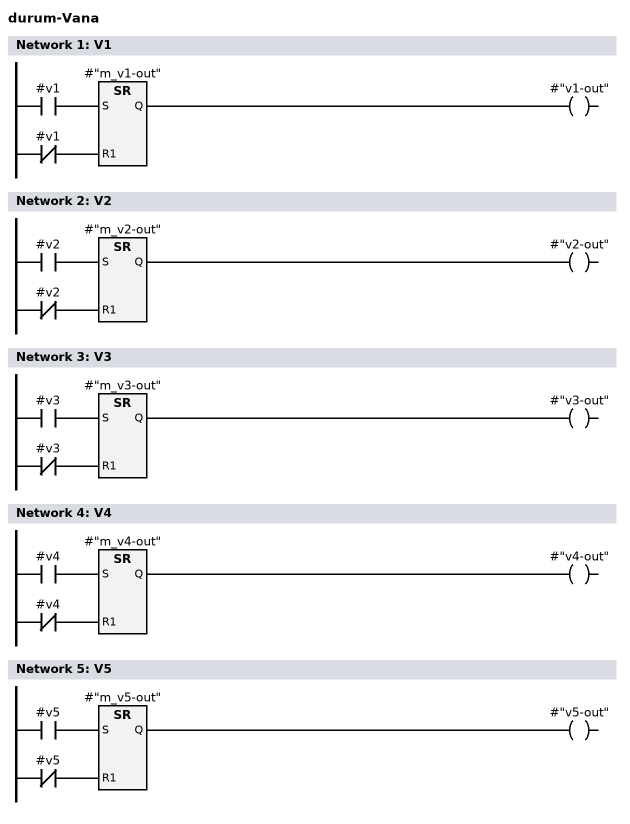
   RUNG wire#powerrail
      Contact( #v1 )
      S_SR(operand := #"m_v1-out", r1 := wire#w1)
      Coil( #"v1-out" )
   END_RUNG
   RUNG wire#powerrail
      I_Contact( #v1 )
   END_RUNG wire#w1
   // the same network as SCL:
   IF #v1 THEN
       #"m_v1-out" := TRUE;   // SR flip-flop
   END_IF;
   IF NOT #v1 THEN #"m_v1-out" := FALSE; END_IF;
   #"v1-out" := #"m_v1-out";
END_REGION

REGION Network 2: V2
   RUNG wire#powerrail
      Contact( #v2 )
      S_SR(operand := #"m_v2-out", r1 := wire#w1)
      Coil( #"v2-out" )
   END_RUNG
   RUNG wire#powerrail
      I_Contact( #v2 )
   END_RUNG wire#w1
   // the same network as SCL:
   IF #v2 THEN
       #"m_v2-out" := TRUE;   // SR flip-flop
   END_IF;
   IF NOT #v2 THEN #"m_v2-out" := FALSE; END_IF;
   #"v2-out" := #"m_v2-out";
END_REGION

REGION Network 3: V3
   RUNG wire#powerrail
      Contact( #v3 )
      S_SR(operand := #"m_v3-out", r1 := wire#w1)
      Coil( #"v3-out" )
   END_RUNG
   RUNG wire#powerrail
      I_Contact( #v3 )
   END_RUNG wire#w1
   // the same network as SCL:
   IF #v3 THEN
       #"m_v3-out" := TRUE;   // SR flip-flop
   END_IF;
   IF NOT #v3 THEN #"m_v3-out" := FALSE; END_IF;
   #"v3-out" := #"m_v3-out";
END_REGION

REGION Network 4: V4
   RUNG wire#powerrail
      Contact( #v4 )
      S_SR(operand := #"m_v4-out", r1 := wire#w1)
      Coil( #"v4-out" )
   END_RUNG
   RUNG wire#powerrail
      I_Contact( #v4 )
   END_RUNG wire#w1
   // the same network as SCL:
   IF #v4 THEN
       #"m_v4-out" := TRUE;   // SR flip-flop
   END_IF;
   IF NOT #v4 THEN #"m_v4-out" := FALSE; END_IF;
   #"v4-out" := #"m_v4-out";
END_REGION

REGION Network 5: V5
   RUNG wire#powerrail
      Contact( #v5 )
      S_SR(operand := #"m_v5-out", r1 := wire#w1)
      Coil( #"v5-out" )
   END_RUNG
   RUNG wire#powerrail
      I_Contact( #v5 )
   END_RUNG wire#w1
   // the same network as SCL:
   IF #v5 THEN
       #"m_v5-out" := TRUE;   // SR flip-flop
   END_IF;
   IF NOT #v5 THEN #"m_v5-out" := FALSE; END_IF;
   #"v5-out" := #"m_v5-out";
END_REGION
END_FUNCTION

ORGANIZATION_BLOCK "Main"   // OB1, LAD, ProgramCycle
TITLE = "Main Program Sweep (Cycle)"
{ S7_Optimized_Access := 'TRUE' }
VERSION : 0.1
   VAR_INPUT
      Initial_Call : Bool;   // Initial call of this OB
      Remanence : Bool;   // =True, if remanent data are available
   END_VAR
   VAR_TEMP
      tempMotorDegis : DInt;
   END_VAR
   VAR CONSTANT
      Constant_1 : Bool;
   END_VAR
   VAR_TEMP   // added for the SCL form of the ladder/FBD networks
      _w1 : Bool;
      _w2 : Bool;
      _w3 : Bool;
      _w4 : Bool;
      _w5 : Bool;
      _w6 : Bool;
   END_VAR
BEGIN

REGION Network 1: Start Stop
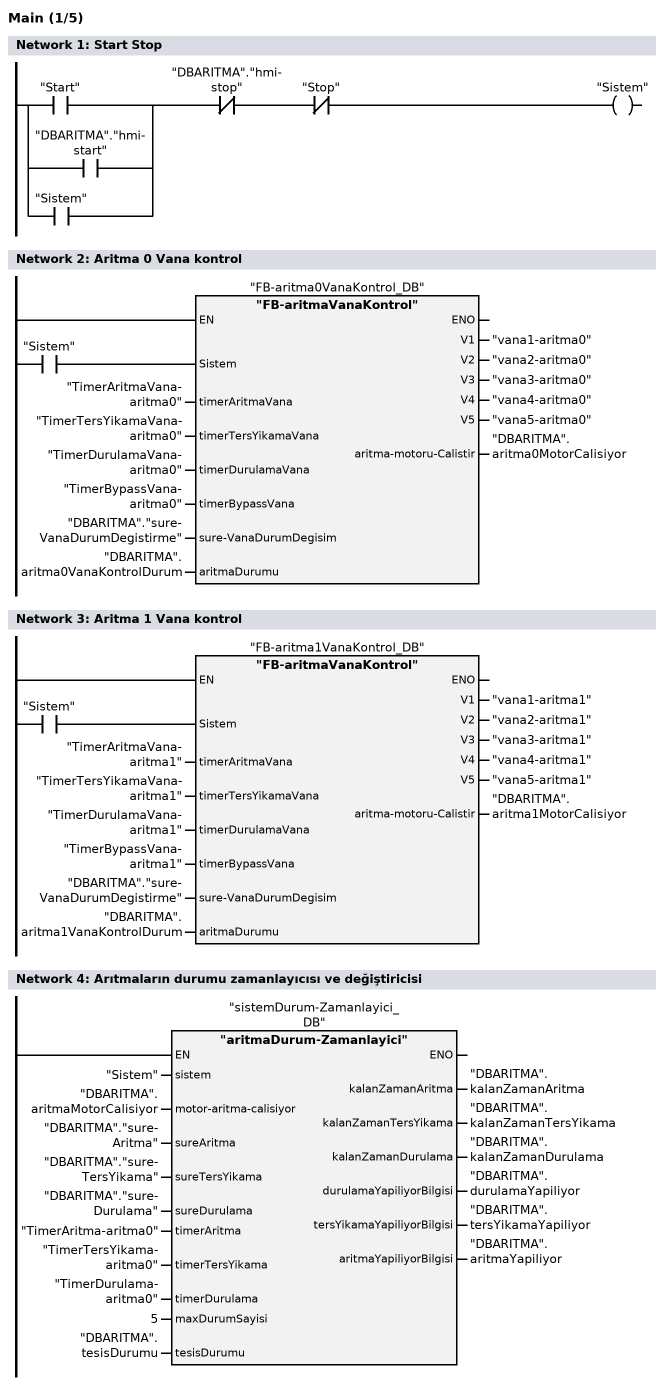
   RUNG wire#powerrail
      Contact( "Start" )
      wire#w1
      I_Contact( "DBARITMA"."hmi-stop" )
      I_Contact( "Stop" )
      Coil( "Sistem" )
   END_RUNG
   RUNG wire#powerrail
      Contact( "DBARITMA"."hmi-start" )
   END_RUNG wire#w1
   RUNG wire#powerrail
      Contact( "Sistem" )
   END_RUNG wire#w1
   // the same network as SCL:
   "Sistem" := ("Start" OR "DBARITMA"."hmi-start" OR "Sistem") AND NOT "DBARITMA"."hmi-stop" AND NOT "Stop";
END_REGION

REGION Network 2: Aritma 0 Vana kontrol
   RUNG wire#powerrail
      "FB-aritma0VanaKontrol_DB"(Sistem := wire#w1, timerAritmaVana := "TimerAritmaVana-aritma0", timerTersYikamaVana := "TimerTersYikamaVana-aritma0", timerDurulamaVana := "TimerDurulamaVana-aritma0", timerBypassVana := "TimerBypassVana-aritma0", "sure-VanaDurumDegisim" := "DBARITMA"."sure-VanaDurumDegistirme", aritmaDurumu := "DBARITMA".aritma0VanaKontrolDurum, V1 => "vana1-aritma0", V2 => "vana2-aritma0", V3 => "vana3-aritma0", V4 => "vana4-aritma0", V5 => "vana5-aritma0", "aritma-motoru-Calistir" => "DBARITMA".aritma0MotorCalisiyor)
   END_RUNG
   RUNG wire#powerrail
      Contact( "Sistem" )
   END_RUNG wire#w1
   // the same network as SCL:
   "FB-aritma0VanaKontrol_DB"(Sistem := "Sistem",   // "FB-aritmaVanaKontrol"
                           timerAritmaVana := "TimerAritmaVana-aritma0",
                           timerTersYikamaVana := "TimerTersYikamaVana-aritma0",
                           timerDurulamaVana := "TimerDurulamaVana-aritma0",
                           timerBypassVana := "TimerBypassVana-aritma0",
                           "sure-VanaDurumDegisim" := "DBARITMA"."sure-VanaDurumDegistirme",
                           aritmaDurumu := "DBARITMA".aritma0VanaKontrolDurum,
                           V1 => "vana1-aritma0",
                           V2 => "vana2-aritma0",
                           V3 => "vana3-aritma0",
                           V4 => "vana4-aritma0",
                           V5 => "vana5-aritma0",
                           "aritma-motoru-Calistir" => "DBARITMA".aritma0MotorCalisiyor);
END_REGION

REGION Network 3: Aritma 1 Vana kontrol
   RUNG wire#powerrail
      "FB-aritma1VanaKontrol_DB"(Sistem := wire#w1, timerAritmaVana := "TimerAritmaVana-aritma1", timerTersYikamaVana := "TimerTersYikamaVana-aritma1", timerDurulamaVana := "TimerDurulamaVana-aritma1", timerBypassVana := "TimerBypassVana-aritma1", "sure-VanaDurumDegisim" := "DBARITMA"."sure-VanaDurumDegistirme", aritmaDurumu := "DBARITMA".aritma1VanaKontrolDurum, V1 => "vana1-aritma1", V2 => "vana2-aritma1", V3 => "vana3-aritma1", V4 => "vana4-aritma1", V5 => "vana5-aritma1", "aritma-motoru-Calistir" => "DBARITMA".aritma1MotorCalisiyor)
   END_RUNG
   RUNG wire#powerrail
      Contact( "Sistem" )
   END_RUNG wire#w1
   // the same network as SCL:
   "FB-aritma1VanaKontrol_DB"(Sistem := "Sistem",   // "FB-aritmaVanaKontrol"
                           timerAritmaVana := "TimerAritmaVana-aritma1",
                           timerTersYikamaVana := "TimerTersYikamaVana-aritma1",
                           timerDurulamaVana := "TimerDurulamaVana-aritma1",
                           timerBypassVana := "TimerBypassVana-aritma1",
                           "sure-VanaDurumDegisim" := "DBARITMA"."sure-VanaDurumDegistirme",
                           aritmaDurumu := "DBARITMA".aritma1VanaKontrolDurum,
                           V1 => "vana1-aritma1",
                           V2 => "vana2-aritma1",
                           V3 => "vana3-aritma1",
                           V4 => "vana4-aritma1",
                           V5 => "vana5-aritma1",
                           "aritma-motoru-Calistir" => "DBARITMA".aritma1MotorCalisiyor);
END_REGION

REGION Network 4: Arıtmaların durumu zamanlayıcısı ve değiştiricisi
   RUNG wire#powerrail
      "sistemDurum-Zamanlayici_DB"(sistem := "Sistem", "motor-aritma-calisiyor" := "DBARITMA".aritmaMotorCalisiyor, sureAritma := "DBARITMA"."sure-Aritma", sureTersYikama := "DBARITMA"."sure-TersYikama", sureDurulama := "DBARITMA"."sure-Durulama", timerAritma := "TimerAritma-aritma0", timerTersYikama := "TimerTersYikama-aritma0", timerDurulama := "TimerDurulama-aritma0", maxDurumSayisi := 5, tesisDurumu := "DBARITMA".tesisDurumu, kalanZamanAritma => "DBARITMA".kalanZamanAritma, kalanZamanTersYikama => "DBARITMA".kalanZamanTersYikama, kalanZamanDurulama => "DBARITMA".kalanZamanDurulama, durulamaYapiliyorBilgisi => "DBARITMA".durulamaYapiliyor, tersYikamaYapiliyorBilgisi => "DBARITMA".tersYikamaYapiliyor, aritmaYapiliyorBilgisi => "DBARITMA".aritmaYapiliyor)
   END_RUNG
   // the same network as SCL:
   "sistemDurum-Zamanlayici_DB"(sistem := "Sistem",   // "aritmaDurum-Zamanlayici"
                           "motor-aritma-calisiyor" := "DBARITMA".aritmaMotorCalisiyor,
                           sureAritma := "DBARITMA"."sure-Aritma",
                           sureTersYikama := "DBARITMA"."sure-TersYikama",
                           sureDurulama := "DBARITMA"."sure-Durulama",
                           timerAritma := "TimerAritma-aritma0",
                           timerTersYikama := "TimerTersYikama-aritma0",
                           timerDurulama := "TimerDurulama-aritma0",
                           maxDurumSayisi := 5,
                           tesisDurumu := "DBARITMA".tesisDurumu,
                           kalanZamanAritma => "DBARITMA".kalanZamanAritma,
                           kalanZamanTersYikama => "DBARITMA".kalanZamanTersYikama,
                           kalanZamanDurulama => "DBARITMA".kalanZamanDurulama,
                           durulamaYapiliyorBilgisi => "DBARITMA".durulamaYapiliyor,
                           tersYikamaYapiliyorBilgisi => "DBARITMA".tersYikamaYapiliyor,
                           aritmaYapiliyorBilgisi => "DBARITMA".aritmaYapiliyor);
END_REGION

REGION Network 5: Aritma motorlarının Eşit Yaşlandırma ve Arıza kontrolü
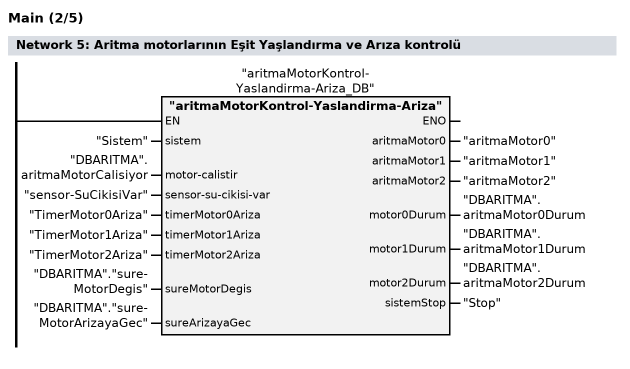
   RUNG wire#powerrail
      "aritmaMotorKontrol-Yaslandirma-Ariza_DB"(sistem := "Sistem", "motor-calistir" := "DBARITMA".aritmaMotorCalisiyor, "sensor-su-cikisi-var" := "sensor-SuCikisiVar", timerMotor0Ariza := "TimerMotor0Ariza", timerMotor1Ariza := "TimerMotor1Ariza", timerMotor2Ariza := "TimerMotor2Ariza", sureMotorDegis := "DBARITMA"."sure-MotorDegis", sureArizayaGec := "DBARITMA"."sure-MotorArizayaGec", aritmaMotor0 => "aritmaMotor0", aritmaMotor1 => "aritmaMotor1", aritmaMotor2 => "aritmaMotor2", motor0Durum => "DBARITMA".aritmaMotor0Durum, motor1Durum => "DBARITMA".aritmaMotor1Durum, motor2Durum => "DBARITMA".aritmaMotor2Durum, sistemStop => "Stop")
   END_RUNG
   // the same network as SCL:
   "aritmaMotorKontrol-Yaslandirma-Ariza_DB"(sistem := "Sistem",   // "aritmaMotorKontrol-Yaslandirma-Ariza"
                           "motor-calistir" := "DBARITMA".aritmaMotorCalisiyor,
                           "sensor-su-cikisi-var" := "sensor-SuCikisiVar",
                           timerMotor0Ariza := "TimerMotor0Ariza",
                           timerMotor1Ariza := "TimerMotor1Ariza",
                           timerMotor2Ariza := "TimerMotor2Ariza",
                           sureMotorDegis := "DBARITMA"."sure-MotorDegis",
                           sureArizayaGec := "DBARITMA"."sure-MotorArizayaGec",
                           aritmaMotor0 => "aritmaMotor0",
                           aritmaMotor1 => "aritmaMotor1",
                           aritmaMotor2 => "aritmaMotor2",
                           motor0Durum => "DBARITMA".aritmaMotor0Durum,
                           motor1Durum => "DBARITMA".aritmaMotor1Durum,
                           motor2Durum => "DBARITMA".aritmaMotor2Durum,
                           sistemStop => "Stop");
END_REGION

REGION Network 6: Arıtma tankları durum kontrolleri
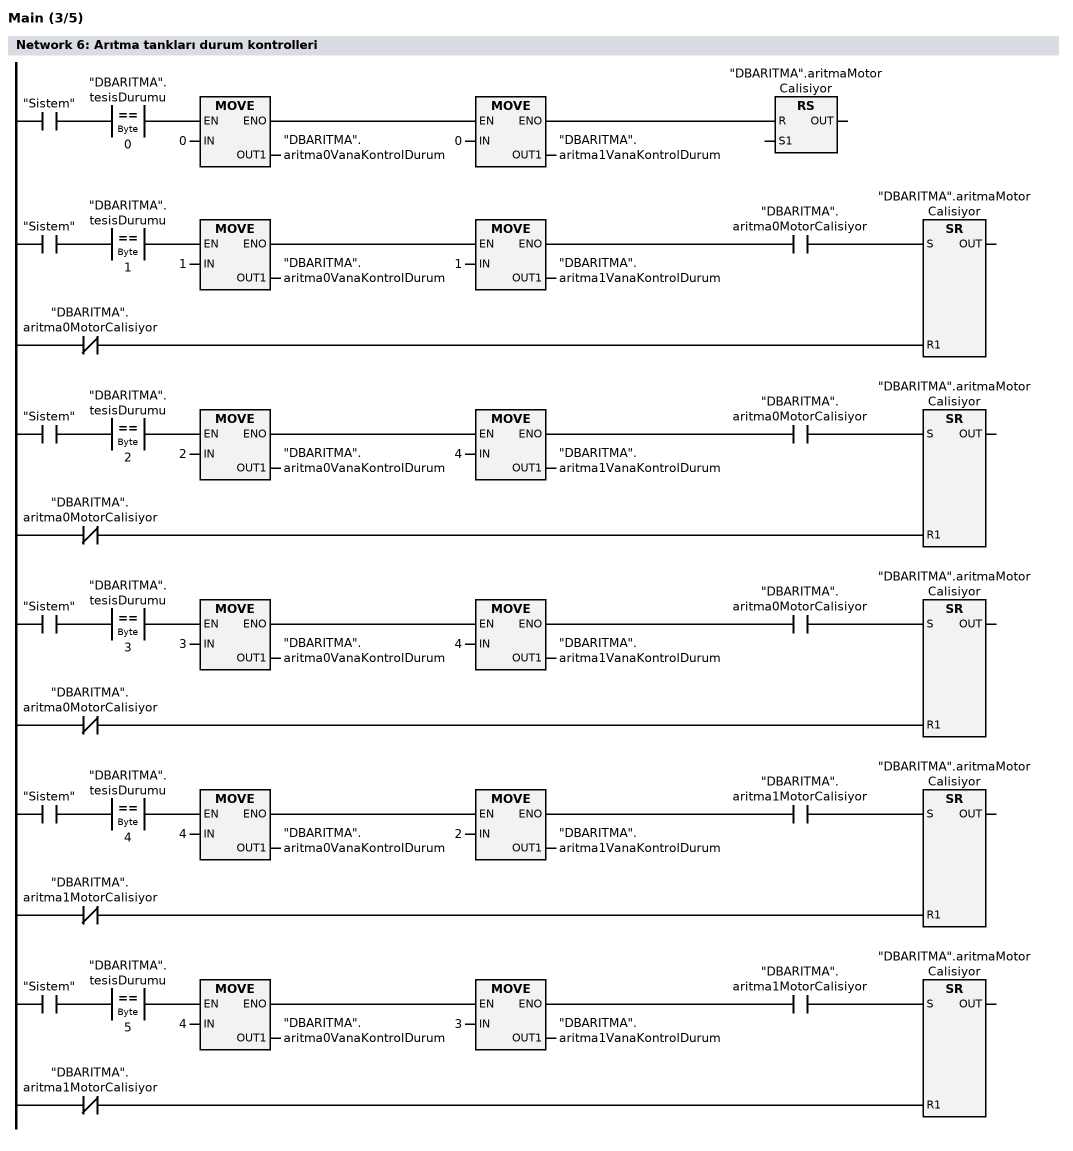
   RUNG wire#powerrail
      Contact( "Sistem" )
      { S7_Templates := "SrcType := Byte" } EQ_Contact(in1 := "DBARITMA".tesisDurumu, in2 := 0)
      Move(in := 0, out1 => "DBARITMA".aritma0VanaKontrolDurum)
      Move(in := 0, out1 => "DBARITMA".aritma1VanaKontrolDurum)
      S_RS(operand := "DBARITMA".aritmaMotorCalisiyor, s1 :=)
   END_RUNG
   RUNG wire#powerrail
      Contact( "Sistem" )
      { S7_Templates := "SrcType := Byte" } EQ_Contact(in1 := "DBARITMA".tesisDurumu, in2 := 1)
      Move(in := 1, out1 => "DBARITMA".aritma0VanaKontrolDurum)
      Move(in := 1, out1 => "DBARITMA".aritma1VanaKontrolDurum)
      Contact( "DBARITMA".aritma0MotorCalisiyor )
      S_SR(operand := "DBARITMA".aritmaMotorCalisiyor, r1 := wire#w1)
   END_RUNG
   RUNG wire#powerrail
      I_Contact( "DBARITMA".aritma0MotorCalisiyor )
   END_RUNG wire#w1
   RUNG wire#powerrail
      Contact( "Sistem" )
      { S7_Templates := "SrcType := Byte" } EQ_Contact(in1 := "DBARITMA".tesisDurumu, in2 := 2)
      Move(in := 2, out1 => "DBARITMA".aritma0VanaKontrolDurum)
      Move(in := 4, out1 => "DBARITMA".aritma1VanaKontrolDurum)
      Contact( "DBARITMA".aritma0MotorCalisiyor )
      S_SR(operand := "DBARITMA".aritmaMotorCalisiyor, r1 := wire#w2)
   END_RUNG
   RUNG wire#powerrail
      I_Contact( "DBARITMA".aritma0MotorCalisiyor )
   END_RUNG wire#w2
   RUNG wire#powerrail
      Contact( "Sistem" )
      { S7_Templates := "SrcType := Byte" } EQ_Contact(in1 := "DBARITMA".tesisDurumu, in2 := 3)
      Move(in := 3, out1 => "DBARITMA".aritma0VanaKontrolDurum)
      Move(in := 4, out1 => "DBARITMA".aritma1VanaKontrolDurum)
      Contact( "DBARITMA".aritma0MotorCalisiyor )
      S_SR(operand := "DBARITMA".aritmaMotorCalisiyor, r1 := wire#w3)
   END_RUNG
   RUNG wire#powerrail
      I_Contact( "DBARITMA".aritma0MotorCalisiyor )
   END_RUNG wire#w3
   RUNG wire#powerrail
      Contact( "Sistem" )
      { S7_Templates := "SrcType := Byte" } EQ_Contact(in1 := "DBARITMA".tesisDurumu, in2 := 4)
      Move(in := 4, out1 => "DBARITMA".aritma0VanaKontrolDurum)
      Move(in := 2, out1 => "DBARITMA".aritma1VanaKontrolDurum)
      Contact( "DBARITMA".aritma1MotorCalisiyor )
      S_SR(operand := "DBARITMA".aritmaMotorCalisiyor, r1 := wire#w4)
   END_RUNG
   RUNG wire#powerrail
      I_Contact( "DBARITMA".aritma1MotorCalisiyor )
   END_RUNG wire#w4
   RUNG wire#powerrail
      Contact( "Sistem" )
      { S7_Templates := "SrcType := Byte" } EQ_Contact(in1 := "DBARITMA".tesisDurumu, in2 := 5)
      Move(in := 4, out1 => "DBARITMA".aritma0VanaKontrolDurum)
      Move(in := 3, out1 => "DBARITMA".aritma1VanaKontrolDurum)
      Contact( "DBARITMA".aritma1MotorCalisiyor )
      S_SR(operand := "DBARITMA".aritmaMotorCalisiyor, r1 := wire#w5)
   END_RUNG
   RUNG wire#powerrail
      I_Contact( "DBARITMA".aritma1MotorCalisiyor )
   END_RUNG wire#w5
   // the same network as SCL:
   #_w1 := "Sistem" AND ("DBARITMA".tesisDurumu = 0);
   IF #_w1 THEN
       "DBARITMA".aritma0VanaKontrolDurum := 0;
       "DBARITMA".aritma1VanaKontrolDurum := 0;
       "DBARITMA".aritmaMotorCalisiyor := FALSE;   // RS flip-flop
   END_IF;
   #_w2 := "Sistem" AND ("DBARITMA".tesisDurumu = 1);
   IF #_w2 THEN
       "DBARITMA".aritma0VanaKontrolDurum := 1;
       "DBARITMA".aritma1VanaKontrolDurum := 1;
   END_IF;
   IF #_w2 AND "DBARITMA".aritma0MotorCalisiyor THEN
       "DBARITMA".aritmaMotorCalisiyor := TRUE;   // SR flip-flop
   END_IF;
   IF NOT "DBARITMA".aritma0MotorCalisiyor THEN "DBARITMA".aritmaMotorCalisiyor := FALSE; END_IF;
   #_w3 := "Sistem" AND ("DBARITMA".tesisDurumu = 2);
   IF #_w3 THEN
       "DBARITMA".aritma0VanaKontrolDurum := 2;
       "DBARITMA".aritma1VanaKontrolDurum := 4;
   END_IF;
   IF #_w3 AND "DBARITMA".aritma0MotorCalisiyor THEN
       "DBARITMA".aritmaMotorCalisiyor := TRUE;   // SR flip-flop
   END_IF;
   IF NOT "DBARITMA".aritma0MotorCalisiyor THEN "DBARITMA".aritmaMotorCalisiyor := FALSE; END_IF;
   #_w4 := "Sistem" AND ("DBARITMA".tesisDurumu = 3);
   IF #_w4 THEN
       "DBARITMA".aritma0VanaKontrolDurum := 3;
       "DBARITMA".aritma1VanaKontrolDurum := 4;
   END_IF;
   IF #_w4 AND "DBARITMA".aritma0MotorCalisiyor THEN
       "DBARITMA".aritmaMotorCalisiyor := TRUE;   // SR flip-flop
   END_IF;
   IF NOT "DBARITMA".aritma0MotorCalisiyor THEN "DBARITMA".aritmaMotorCalisiyor := FALSE; END_IF;
   #_w5 := "Sistem" AND ("DBARITMA".tesisDurumu = 4);
   IF #_w5 THEN
       "DBARITMA".aritma0VanaKontrolDurum := 4;
       "DBARITMA".aritma1VanaKontrolDurum := 2;
   END_IF;
   IF #_w5 AND "DBARITMA".aritma1MotorCalisiyor THEN
       "DBARITMA".aritmaMotorCalisiyor := TRUE;   // SR flip-flop
   END_IF;
   IF NOT "DBARITMA".aritma1MotorCalisiyor THEN "DBARITMA".aritmaMotorCalisiyor := FALSE; END_IF;
   #_w6 := "Sistem" AND ("DBARITMA".tesisDurumu = 5);
   IF #_w6 THEN
       "DBARITMA".aritma0VanaKontrolDurum := 4;
       "DBARITMA".aritma1VanaKontrolDurum := 3;
   END_IF;
   IF #_w6 AND "DBARITMA".aritma1MotorCalisiyor THEN
       "DBARITMA".aritmaMotorCalisiyor := TRUE;   // SR flip-flop
   END_IF;
   IF NOT "DBARITMA".aritma1MotorCalisiyor THEN "DBARITMA".aritmaMotorCalisiyor := FALSE; END_IF;
END_REGION

REGION Network 7: Temizsu depo seviyesine göre arıtma işlemini başlat
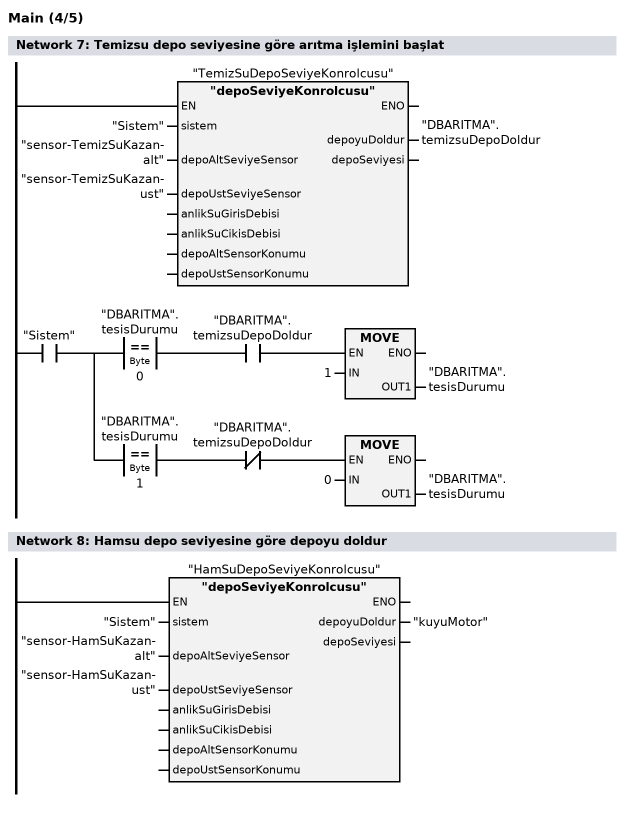
   RUNG wire#powerrail
      "TemizSuDepoSeviyeKonrolcusu"(sistem := "Sistem", depoAltSeviyeSensor := "sensor-TemizSuKazan-alt", depoUstSeviyeSensor := "sensor-TemizSuKazan-ust", anlikSuGirisDebisi :=, anlikSuCikisDebisi :=, depoAltSensorKonumu :=, depoUstSensorKonumu :=, depoyuDoldur => "DBARITMA".temizsuDepoDoldur, depoSeviyesi =>)
   END_RUNG
   RUNG wire#powerrail
      Contact( "Sistem" )
      wire#w1
      { S7_Templates := "SrcType := Byte" } EQ_Contact(in1 := "DBARITMA".tesisDurumu, in2 := 0)
      Contact( "DBARITMA".temizsuDepoDoldur )
      Move(in := 1, out1 => "DBARITMA".tesisDurumu)
   END_RUNG
   RUNG wire#w1
      { S7_Templates := "SrcType := Byte" } EQ_Contact(in1 := "DBARITMA".tesisDurumu, in2 := 1)
      I_Contact( "DBARITMA".temizsuDepoDoldur )
      Move(in := 0, out1 => "DBARITMA".tesisDurumu)
   END_RUNG
   // the same network as SCL:
   "TemizSuDepoSeviyeKonrolcusu"(sistem := "Sistem",   // "depoSeviyeKonrolcusu"
                           depoAltSeviyeSensor := "sensor-TemizSuKazan-alt",
                           depoUstSeviyeSensor := "sensor-TemizSuKazan-ust",
                           depoyuDoldur => "DBARITMA".temizsuDepoDoldur);
   IF "Sistem" AND ("DBARITMA".tesisDurumu = 0) AND "DBARITMA".temizsuDepoDoldur THEN
       "DBARITMA".tesisDurumu := 1;
   END_IF;
   IF "Sistem" AND ("DBARITMA".tesisDurumu = 1) AND NOT "DBARITMA".temizsuDepoDoldur THEN
       "DBARITMA".tesisDurumu := 0;
   END_IF;
END_REGION

REGION Network 8: Hamsu depo seviyesine göre depoyu doldur
   RUNG wire#powerrail
      "HamSuDepoSeviyeKonrolcusu"(sistem := "Sistem", depoAltSeviyeSensor := "sensor-HamSuKazan-alt", depoUstSeviyeSensor := "sensor-HamSuKazan-ust", anlikSuGirisDebisi :=, anlikSuCikisDebisi :=, depoAltSensorKonumu :=, depoUstSensorKonumu :=, depoyuDoldur => "kuyuMotor", depoSeviyesi =>)
   END_RUNG
   // the same network as SCL:
   "HamSuDepoSeviyeKonrolcusu"(sistem := "Sistem",   // "depoSeviyeKonrolcusu"
                           depoAltSeviyeSensor := "sensor-HamSuKazan-alt",
                           depoUstSeviyeSensor := "sensor-HamSuKazan-ust",
                           depoyuDoldur => "kuyuMotor");
END_REGION

REGION Network 9: Hmi ayarları
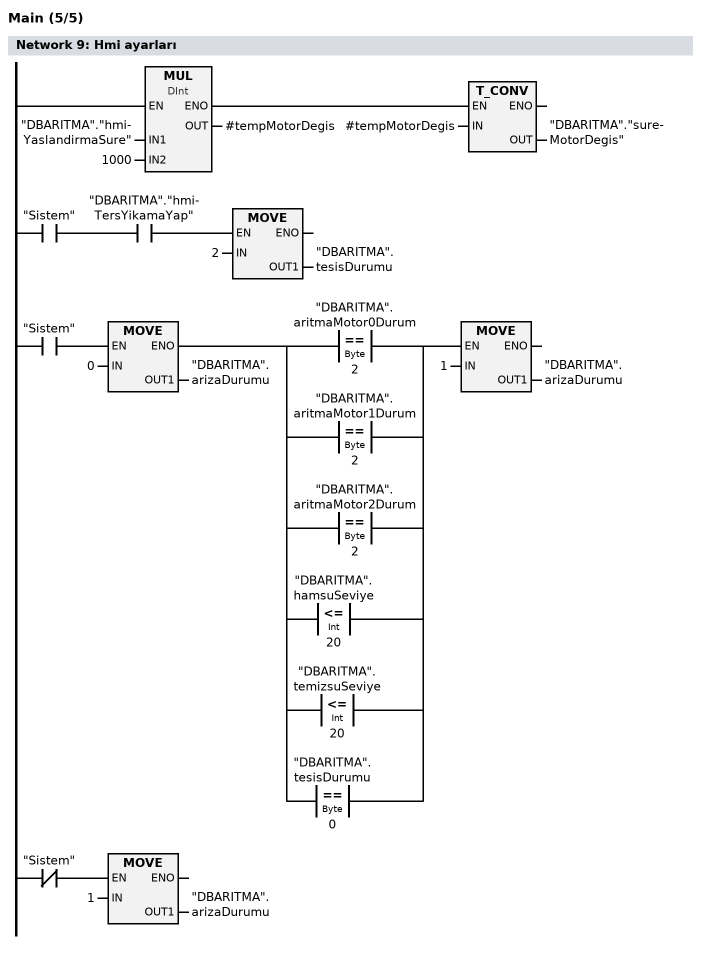
   #tempMotorDegis := "DBARITMA"."hmi-YaslandirmaSure" * 1000;
   "DBARITMA"."sure-MotorDegis" := T_CONV(IN := #tempMotorDegis);
   IF "Sistem" AND "DBARITMA"."hmi-TersYikamaYap" THEN "DBARITMA".tesisDurumu := 2; END_IF;
   IF "Sistem" THEN "DBARITMA".arizaDurumu := 0; END_IF;
   IF "Sistem" AND (("DBARITMA".aritmaMotor0Durum = 2) OR ("DBARITMA".aritmaMotor1Durum = 2) OR ("DBARITMA".aritmaMotor2Durum = 2) OR ("DBARITMA".hamsuSeviye <= 20) OR ("DBARITMA".temizsuSeviye <= 20) OR ("DBARITMA".tesisDurumu = 0)) THEN
       "DBARITMA".arizaDurumu := 1;
   END_IF;
   IF NOT "Sistem" THEN "DBARITMA".arizaDurumu := 1; END_IF;
END_REGION
END_ORGANIZATION_BLOCK

(* ===== HMI "HMI_RT_1" =====
system functions are stored by id; their names below are inferred from use
connection "HMI_Connection_1": ETHERNET, SMART_S7_1500_OMS

HMI tags "Default tag table"
   "aritmaMotor0" : Bool = PLC aritmaMotor0 AT %Q0.0, 100 ms
   "vana1-aritma0" : Bool = PLC "vana1-aritma0" AT %Q0.4, 100 ms
   "vana2-aritma0" : Bool = PLC "vana2-aritma0" AT %Q0.5, 100 ms
   "vana3-aritma0" : Bool = PLC "vana3-aritma0" AT %Q0.6, 100 ms
   "vana4-aritma0" : Bool = PLC "vana4-aritma0" AT %Q0.7, 100 ms
   "vana5-aritma0" : Bool = PLC "vana5-aritma0" AT %Q1.0, 100 ms
   "Start" : Bool = PLC Start AT %I0.0, 100 ms
   "Stop" : Bool = PLC Stop AT %I0.1, 100 ms
   "Sistem" : Bool = PLC Sistem AT %Q1.6, 100 ms
   "DBARITMA_durum-Sistem" : Byte = PLC DBARITMA.tesisDurumu AT %DB1.DBB14, 100 ms
   "DBARITMA_aritmaMotorCalisiyor" : Bool = PLC DBARITMA.aritmaMotorCalisiyor AT %DB1.DBX18.2, 100 ms
   "DBARITMA_aritmaYapiliyor" : Bool = PLC DBARITMA.aritmaYapiliyor AT %DB1.DBX26.0, 100 ms
   "DBARITMA_tersYikamaYapiliyor" : Bool = PLC DBARITMA.tersYikamaYapiliyor AT %DB1.DBX26.1, 100 ms
   "DBARITMA_durulamaYapiliyor" : Bool = PLC DBARITMA.durulamaYapiliyor AT %DB1.DBX26.2, 100 ms
   "DBARITMA_kalanZamanAritma" : S5Time = PLC DBARITMA.kalanZamanAritma AT %DB1.DBW20, 100 ms
   "DBARITMA_kalanZamanTersYikama" : S5Time = PLC DBARITMA.kalanZamanTersYikama AT %DB1.DBW22, 100 ms
   "DBARITMA_kalanZamanDurulama" : S5Time = PLC DBARITMA.kalanZamanDurulama AT %DB1.DBW24, 100 ms
   "TimerAritma" : Timer = PLC "TimerAritma-aritma0" AT %T18, 100 ms
   "TimerTersYikama" : Timer = PLC "TimerTersYikama-aritma0" AT %T10, 100 ms
   "TimerDurulama" : Timer = PLC "TimerDurulama-aritma0" AT %T11, 100 ms
   "aritmaMotor1" : Bool = PLC aritmaMotor1 AT %Q0.1, 100 ms
   "aritmaMotor2" : Bool = PLC aritmaMotor2 AT %Q0.2, 100 ms
   "sensor-SuCikisiVar" : Bool = PLC "sensor-SuCikisiVar" AT %I0.6, 100 ms
   "timerMotorDegistirme_ET" : Time = PLC timerMotorDegistirme.ET, 100 ms
   "vana1-aritma1" : Bool = PLC "vana1-aritma1" AT %Q1.1, 100 ms
   "vana2-aritma1" : Bool = PLC "vana2-aritma1" AT %Q1.2, 100 ms
   "vana3-aritma1" : Bool = PLC "vana3-aritma1" AT %Q1.3, 100 ms
   "vana4-aritma1" : Bool = PLC "vana4-aritma1" AT %Q1.4, 100 ms
   "vana5-aritma1" : Bool = PLC "vana5-aritma1" AT %Q1.5, 100 ms
   "sensor-HamSuKazan-alt" : Bool = PLC "sensor-HamSuKazan-alt" AT %I0.2, 100 ms
   "sensor-HamSuKazan-ust" : Bool = PLC "sensor-HamSuKazan-ust" AT %I0.3, 100 ms
   "sensor-TemizSuKazan-alt" : Bool = PLC "sensor-TemizSuKazan-alt" AT %I0.4, 100 ms
   "sensor-TemizSuKazan-ust" : Bool = PLC "sensor-TemizSuKazan-ust" AT %I0.5, 100 ms
   "kuyuMotor" : Bool = PLC kuyuMotor AT %I0.7, 100 ms
   "DBARITMA_aritmaMotor0Durum" : Byte = PLC DBARITMA.aritmaMotor0Durum AT %DB1.DBB27, 1 s
   "DBARITMA_aritma1MotorCalisiyor" : Bool = PLC DBARITMA.aritma1MotorCalisiyor AT %DB1.DBX18.1, 1 s
   "DBARITMA_aritmaMotor1Durum" : Byte = PLC DBARITMA.aritmaMotor1Durum AT %DB1.DBB28, 1 s
   "DBARITMA_aritmaMotor2Durum" : Byte = PLC DBARITMA.aritmaMotor2Durum AT %DB1.DBB29, 1 s
   "DBARITMA_hmi-start" : Bool = PLC DBARITMA.hmi-start AT %DB1.DBX294.1, 1 s
   "DBARITMA_hmi-stop" : Bool = PLC DBARITMA.hmi-stop AT %DB1.DBX294.2, 1 s
   "DBARITMA_sure-Aritma" : S5Time = PLC DBARITMA.sure-Aritma AT %DB1.DBW0, 1 s
   "DBARITMA_sure-MotorDegis" : Time = PLC DBARITMA.sure-MotorDegis AT %DB1.DBD8, 1 s
   "DBARITMA_hmi-aritmaSure" : Byte = PLC DBARITMA.hmi-aritmaSure AT %DB1.DBB295, 1 s
   "DBARITMA_hmi-YaslandirmaSure" : Byte = PLC DBARITMA.hmi-YaslandirmaSure AT %DB1.DBB299, 1 s
   "DBARITMA_hmi-TersYikamaYap" : Bool = PLC DBARITMA.hmi-TersYikamaYap AT %DB1.DBX300.0, 1 s
   "DBARITMA_kuyuMotorDurum" : Byte = PLC DBARITMA.kuyuMotorDurum AT %DB1.DBB30, 1 s

discrete alarms
   1: '', class Errors
   2: '', class Acknowledgement bit 0
   3: '', class No Acknowledgement bit 0

screen "aritma-ekrani" 800x480
   Button "btn-aritmaEkraniGeri" at 5,431 size 112x43; TextOff 'GERİ'
      on Press: function_efd93a16()
   TextField "Text field_1" at 261,15 size 152x25; Text 'DEMİR ARITMA'
   TextField "Text field_2" at 605,13 size 173x25; Text 'MANGAN ARITMA'
   TextField "Text field_3" at 118,131 size 26x23; Text 'V1'
   TextField "Text field_5" at 198,307 size 26x23; Text 'V5'
   TextField "Text field_6" at 118,273 size 26x23; Text 'V3'
   TextField "Text field_7" at 97,307 size 26x23; Text 'V2'
   TextField "Text field_10" at 485,273 size 26x23; Text 'V3'
   GraphicView "Graphic view_3" at 262,337 size 39x37; Picture "Graphic_14"
   GraphicView "Graphic view_1" at 634,337 size 39x37; Picture "Graphic_14"
   TextField "Text field_13" at 670,423 size 127x40; Text 'TEMİZ SU DEPO BAĞLANTISI'
   Switch "Switch_1" at 14,40 size 64x32; CaptionText 'Switch'; TextOff 'OFF'; TextOn 'ON'
      on SwitchOn: SetBit("sensor-SuCikisiVar")
      on SwitchOff: ResetBit("sensor-SuCikisiVar")
      ProcessValue <- "sensor-SuCikisiVar"
   TextField "Text field_14" at 1,99 size 68x23; Text 'Motor 1'
   TextField "Text field_15" at 1,246 size 68x23; Text 'Motor 3'
   TextField "Text field_16" at 1,172 size 68x23; Text 'Motor 2'
   TextField "Text field_17" at 14,7 size 138x23; Text 'Arıtma Yapılıyor'
      Visibility <- "DBARITMA_aritmaYapiliyor"
      Appearance <- "DBARITMA_aritmaYapiliyor"
   TextField "Text field_18" at 14,7 size 184x23; Text 'Ters Yıkama Yapılıyor'
      Visibility <- "DBARITMA_tersYikamaYapiliyor"
      Appearance <- "DBARITMA_tersYikamaYapiliyor"
   TextField "Text field_21" at 14,7 size 161x23; Text 'Durulama Yapılıyor'
      Visibility <- "DBARITMA_durulamaYapiliyor"
      Appearance <- "DBARITMA_durulamaYapiliyor"
   Button "btn-aritmaEkraniGeri_1" at 325,431 size 160x43; TextOff 'ARITMA AYARLARI'
      on Press: ActivateScreen("aritma-ayarlari", 0)
   Button "btn-aritmaEkraniGeri_2" at 512,431 size 150x43; TextOff 'TERS YIKAMA YAP'
      on Press: function_b14e0dd5("DBARITMA_hmi-TersYikamaYap", 0)
   Button "btn-aritmaEkraniGeri_3" at 141,431 size 158x43; TextOff 'ARITMA BİLGİLERİ'
      on Press: function_efd93a16()
   Switch "Switch_2" at 401,70 size 64x32; TextOn 'ON'; CaptionText 'Switch'; TextOff 'OFF'
      on SwitchOff: ResetBit("sensor-TemizSuKazan-ust")
      on SwitchOn: SetBit("sensor-TemizSuKazan-ust")
      ProcessValue <- "sensor-TemizSuKazan-ust"
   Switch "Switch_3" at 401,139 size 64x32; TextOn 'ON'; CaptionText 'Switch'; TextOff 'OFF'
      on SwitchOff: ResetBit("sensor-TemizSuKazan-alt")
      on SwitchOn: SetBit("sensor-TemizSuKazan-alt")
      ProcessValue <- "sensor-TemizSuKazan-alt"
   TextField "Text field_19" at 390,49 size 86x22; Text 'Üst Sensör'
   TextField "Text field_20" at 393,118 size 82x22; Text 'Alt Sensör'
   GraphicView "aritma-motor0-ready" at 2,120 size 60x40; Picture "Graphic_37"
      Visibility <- "DBARITMA_aritmaMotor0Durum"
   GraphicView "Graphic view_2" at 2,193 size 60x40; Picture "Graphic_37"
      Visibility <- "DBARITMA_aritmaMotor1Durum"
   GraphicView "aritma-motor1-on" at 2,193 size 60x40; Picture "Graphic_38"
      Visibility <- "DBARITMA_aritmaMotor1Durum"
   GraphicView "aritma-motor0-on" at 2,120 size 60x40; Picture "Graphic_38"
      Visibility <- "DBARITMA_aritmaMotor0Durum"
   GraphicView "aritma-motor0-broken" at 2,120 size 60x40; Picture "Graphic_36"
      Visibility <- "DBARITMA_aritmaMotor0Durum"
   GraphicView "aritma-motor1-broken" at 2,193 size 60x40; Picture "Graphic_36"
      Visibility <- "DBARITMA_aritmaMotor1Durum"
   GraphicView "aritma-motor2-ready" at 2,266 size 60x40; Picture "Graphic_37"
      Visibility <- "DBARITMA_aritmaMotor2Durum"
   GraphicView "aritma-motor2-on" at 2,266 size 60x40; Picture "Graphic_38"
      Visibility <- "DBARITMA_aritmaMotor2Durum"
   GraphicView "aritma-motor2-broken" at 2,266 size 60x40; Picture "Graphic_36"
      Visibility <- "DBARITMA_aritmaMotor2Durum"
   TextField "Text field_8" at 485,131 size 26x23; Text 'V1'
   GraphicView "aritma1vana1-on" at 511,122 size 34x41; Picture "Graphic_47"
      Visibility <- "vana1-aritma1"
   GraphicView "aritma1vana1-off" at 511,122 size 34x41; Picture "Graphic_48"
      Visibility <- "vana1-aritma1"
   TextField "Text field_9" at 565,115 size 26x23; Text 'V4'
   GraphicView "aritma1vana4-off" at 558,84 size 41x34; Picture "Graphic_46"
      Visibility <- "vana4-aritma1"
   GraphicView "aritma1vana4-on" at 558,84 size 41x34; Picture "Graphic_45"
      Visibility <- "vana4-aritma1"
   GraphicView "aritma1vana3-on" at 511,263 size 34x41; Picture "Graphic_47"
      Visibility <- "vana3-aritma1"
   GraphicView "aritma1vana3-off" at 511,263 size 34x41; Picture "Graphic_48"
      Visibility <- "vana3-aritma1"
   TextField "Text field_11" at 462,307 size 26x23; Text 'V2'
   GraphicView "aritma1vana2-off" at 456,331 size 41x34; Picture "Graphic_46"
      Visibility <- "vana2-aritma1"
   GraphicView "aritma1vana2-on" at 456,331 size 41x34; Picture "Graphic_45"
      Visibility <- "vana2-aritma1"
   TextField "Text field_12" at 565,307 size 26x23; Text 'V5'
   GraphicView "aritma1vana5" at 559,332 size 41x34; Picture "Graphic_46"
      Visibility <- "vana5-aritma1"
   GraphicView "aritma1vana5-on" at 559,332 size 41x34; Picture "Graphic_45"
      Visibility <- "vana5-aritma1"
   TextField "Text field_4" at 198,115 size 26x23; Text 'V4'
   GraphicView "aritma0vana4-off" at 191,84 size 41x34; Picture "Graphic_46"
      Visibility <- "vana4-aritma0"
   GraphicView "aritma0vana4-on" at 191,84 size 41x34; Picture "Graphic_45"
      Visibility <- "vana4-aritma0"
   GraphicView "aritma0vana1-on" at 144,122 size 34x41; Picture "Graphic_47"
      Visibility <- "vana1-aritma0"
   GraphicView "aritma0vana1-off" at 144,122 size 34x41; Picture "Graphic_48"
      Visibility <- "vana1-aritma0"
   GraphicView "aritma0vana3-on" at 144,263 size 34x41; Picture "Graphic_47"
      Visibility <- "vana3-aritma0"
   GraphicView "aritma0vana3-off" at 144,263 size 34x41; Picture "Graphic_48"
      Visibility <- "vana3-aritma0"
   GraphicView "aritma0vana2-on" at 89,331 size 41x34; Picture "Graphic_45"
      Visibility <- "vana2-aritma0"
   GraphicView "aritma0vana2-off" at 89,331 size 41x34; Picture "Graphic_46"
      Visibility <- "vana2-aritma0"
   GraphicView "aritma0vana5-on" at 192,332 size 41x34; Picture "Graphic_45"
      Visibility <- "vana5-aritma0"
   GraphicView "aritma0vana5-off" at 192,332 size 41x34; Picture "Graphic_46"
      Visibility <- "vana5-aritma0"
   GraphicView "demir-aritmatank" at 286,78 size 83x243; Picture "Graphic_20"
   GraphicView "demir-aritmatank_1" at 653,78 size 83x243; Picture "Graphic_20"

screen "giris-ekrani" 800x480, template "Template_1"
   GraphicView "Graphic view_1" at 10,22 size 136x140; Picture "aydın bşb"
   GraphicView "Graphic view_2" at 660,6 size 123x159; Picture "logo"
   TextField "Text field_1" at 239,0 size 353x170; Text 'AYDIN BÜYÜKŞEHİR BELEDİYESİ ASKİ GENEL MÜDÜRLÜĞÜ'
   Button "btn-hamkuyusayfa" at 50,404 size 154x64; TextOff 'KUYU HAMSU DEPOSU'
      on Press: ActivateScreen("kuyu-hamsu-ekran", 0)
   Button "btn-aritmasayfa" at 597,404 size 154x64; TextOff 'ARITMA TESİSİ TEMİZSU DEPOSU'
      on Press: ActivateScreen("aritma-ekrani", 0)
   GraphicView "Graphic view_4" at 49,172 size 151x228; Picture "Graphic_6"
   GraphicView "Graphic view_3" at 600,172 size 151x228; Picture "Graphic_6"
   Bar "Bar_1" at 80,209 size 88x129; MinimumValue 0; MaximumValue 100
   Bar "Bar_2" at 632,211 size 88x129; MinimumValue 0; MaximumValue 100
   Button "btn-start" at 252,186 size 112x58; TextOff 'START'
      on Press: function_b14e0dd5("Start", 0)
   Button "btn-stop" at 434,186 size 112x58; TextOff 'STOP'
      on Press: function_b14e0dd5("DBARITMA_hmi-stop", 0)
   Circle "Circle_1" at 375,127 size 48x48
      Appearance <- "Sistem"
   TextField "Text field_2" at 312,89 size 190x29; Text 'SİSTEM DURUMU'

screen "kuyu-hamsu-ekran" 800x480
   GraphicView "Graphic view_3" at 160,265 size 130x120; Picture "Graphic_12"
      Visibility <- "kuyuMotor"
   GraphicView "Graphic view_1" at 216,89 size 130x120; Picture "Graphic_10"
      Visibility <- "DBARITMA_kuyuMotorDurum"
   GraphicView "Graphic view_2" at 159,266 size 130x120; Picture "Graphic_11"
      Visibility <- "kuyuMotor"
   GraphicView "Graphic view_9" at 510,114 size 231x361; Picture "Graphic_20"
   Bar "Bar_1" at 568,179 size 122x198; MinimumValue 0; MaximumValue 100
   Button "btn-aritmaEkraniGeri" at 5,398 size 148x76; TextOff 'GERİ'
      on Press: function_efd93a16()
   TextField "Text field_6" at 67,20 size 224x43; Text 'KUYU HAMSU'
   Button "btn-aritmaEkraniGeri_1" at 5,124 size 148x76; TextOff 'KUYU BİLGİLERİ'
      on Press: function_efd93a16()
   Switch "Switch_1" at 305,430 size 64x32; CaptionText 'Switch'; TextOff 'OFF'; TextOn 'ON'
      ProcessValue <- "sensor-HamSuKazan-alt"
      on SwitchOn: SetBit("sensor-HamSuKazan-alt")
      on SwitchOff: ResetBit("sensor-HamSuKazan-alt")
   TextField "Text field_1" at 389,431 size 93x25; Text 'Alt Sensör'
   Switch "Switch_2" at 305,390 size 64x32; TextOn 'ON'; CaptionText 'Switch'; TextOff 'OFF'
      on SwitchOn: SetBit("sensor-HamSuKazan-ust")
      on SwitchOff: ResetBit("sensor-HamSuKazan-ust")
      ProcessValue <- "sensor-HamSuKazan-ust"
   TextField "Text field_2" at 389,391 size 98x25; Text 'Üst Sensör'

screen "aritma-ayarlari" 800x480, template "Template_1"
   TextField "Text field_1" at 76,117 size 249x29; Text 'Arıtma Süresi(Saniye):'
   TextField "Text field_2" at 76,159 size 308x29; Text 'Ters Yıkama Süresi(Saniye):'
   TextField "Text field_3" at 76,204 size 281x29; Text 'Durulama Süresi(Saniye):'
   TextField "Text field_4" at 76,312 size 326x29; Text 'Vana Bekleme Süresi(Saniye):'
   TextField "Text field_5" at 76,351 size 468x29; Text 'Motor Yaşlandırma Değişim Süresi(Saniye):'
   TextField "Text field_6" at 174,20 size 471x43; Text 'ARITMA BÖLÜMÜ AYARLARI'
   Button "btn-aritmaEkraniGeri" at 5,431 size 148x43; TextOff 'GERİ'
      on Press: function_efd93a16()
   IOField "I/O field_2" at 542,351 size 96x32; FormatPattern 999
      ProcessValue <- "DBARITMA_hmi-YaslandirmaSure"
   TextField "Text field_7" at 323,117 size 35x32; Text '60'
   TextField "Text field_8" at 384,159 size 35x32; Text '20'
   TextField "Text field_9" at 357,203 size 35x32; Text '10'
   TextField "Text field_10" at 405,309 size 20x32; Text '5'
*)